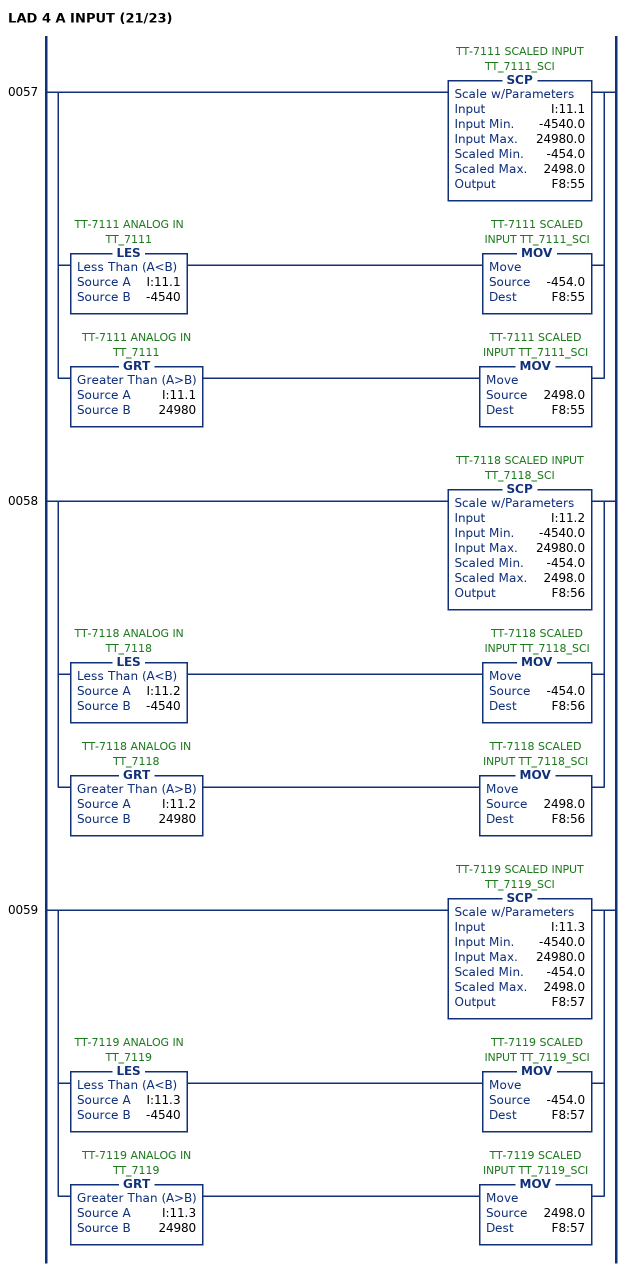
% Rung: 57 %
SOR BST SCP I:11.1 -4540.0 24980.0 -454.0 2498.0 F8:55 NXB LES I:11.1 -4540 MOV -454.0 F8:55 NXB GRT I:11.1 24980 MOV 2498.0 F8:55 BND EOR
%   I:11.1  TT_7111  "TT-7111 ANALOG IN" %
%   F8:55  TT_7111_SCI  "TT-7111 SCALED INPUT" %
% Rung: 58 %
SOR BST SCP I:11.2 -4540.0 24980.0 -454.0 2498.0 F8:56 NXB LES I:11.2 -4540 MOV -454.0 F8:56 NXB GRT I:11.2 24980 MOV 2498.0 F8:56 BND EOR
%   I:11.2  TT_7118  "TT-7118 ANALOG IN" %
%   F8:56  TT_7118_SCI  "TT-7118 SCALED INPUT" %
% Rung: 59 %
SOR BST SCP I:11.3 -4540.0 24980.0 -454.0 2498.0 F8:57 NXB LES I:11.3 -4540 MOV -454.0 F8:57 NXB GRT I:11.3 24980 MOV 2498.0 F8:57 BND EOR
%   I:11.3  TT_7119  "TT-7119 ANALOG IN" %
%   F8:57  TT_7119_SCI  "TT-7119 SCALED INPUT" %

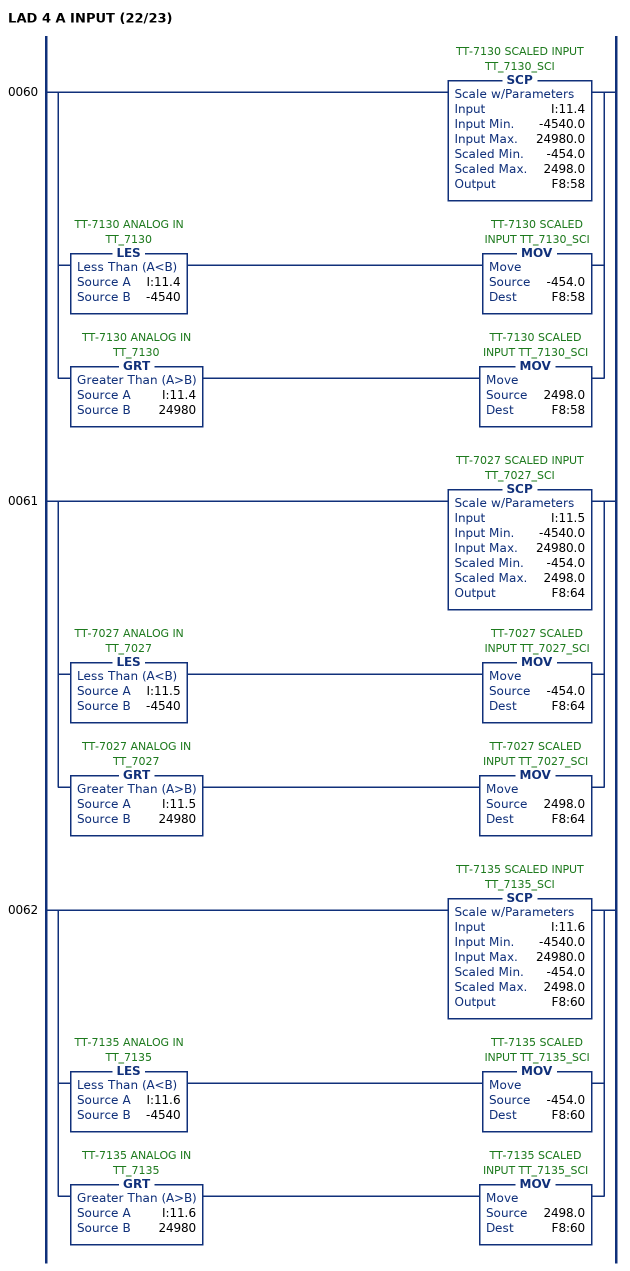
% Rung: 60 %
SOR BST SCP I:11.4 -4540.0 24980.0 -454.0 2498.0 F8:58 NXB LES I:11.4 -4540 MOV -454.0 F8:58 NXB GRT I:11.4 24980 MOV 2498.0 F8:58 BND EOR
%   I:11.4  TT_7130  "TT-7130 ANALOG IN" %
%   F8:58  TT_7130_SCI  "TT-7130 SCALED INPUT" %
% Rung: 61 %
SOR BST SCP I:11.5 -4540.0 24980.0 -454.0 2498.0 F8:64 NXB LES I:11.5 -4540 MOV -454.0 F8:64 NXB GRT I:11.5 24980 MOV 2498.0 F8:64 BND EOR
%   I:11.5  TT_7027  "TT-7027 ANALOG IN" %
%   F8:64  TT_7027_SCI  "TT-7027 SCALED INPUT" %
% Rung: 62 %
SOR BST SCP I:11.6 -4540.0 24980.0 -454.0 2498.0 F8:60 NXB LES I:11.6 -4540 MOV -454.0 F8:60 NXB GRT I:11.6 24980 MOV 2498.0 F8:60 BND EOR
%   I:11.6  TT_7135  "TT-7135 ANALOG IN" %
%   F8:60  TT_7135_SCI  "TT-7135 SCALED INPUT" %

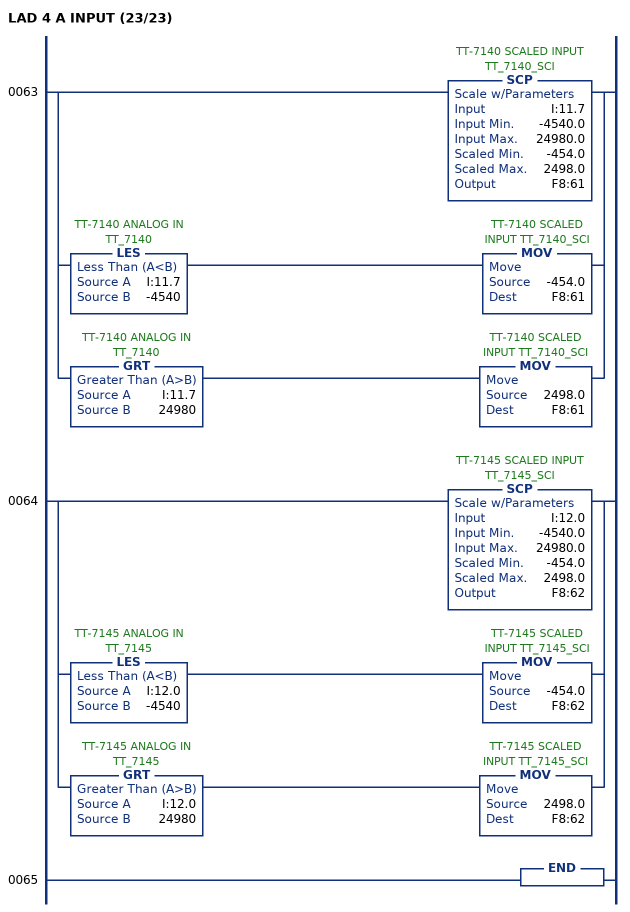
% Rung: 63 %
SOR BST SCP I:11.7 -4540.0 24980.0 -454.0 2498.0 F8:61 NXB LES I:11.7 -4540 MOV -454.0 F8:61 NXB GRT I:11.7 24980 MOV 2498.0 F8:61 BND EOR
%   I:11.7  TT_7140  "TT-7140 ANALOG IN" %
%   F8:61  TT_7140_SCI  "TT-7140 SCALED INPUT" %
% Rung: 64 %
SOR BST SCP I:12.0 -4540.0 24980.0 -454.0 2498.0 F8:62 NXB LES I:12.0 -4540 MOV -454.0 F8:62 NXB GRT I:12.0 24980 MOV 2498.0 F8:62 BND EOR
%   I:12.0  TT_7145  "TT-7145 ANALOG IN" %
%   F8:62  TT_7145_SCI  "TT-7145 SCALED INPUT" %
% Rung: 65 %
SOR END EOR

LADDER 5 "D OUTPUT"
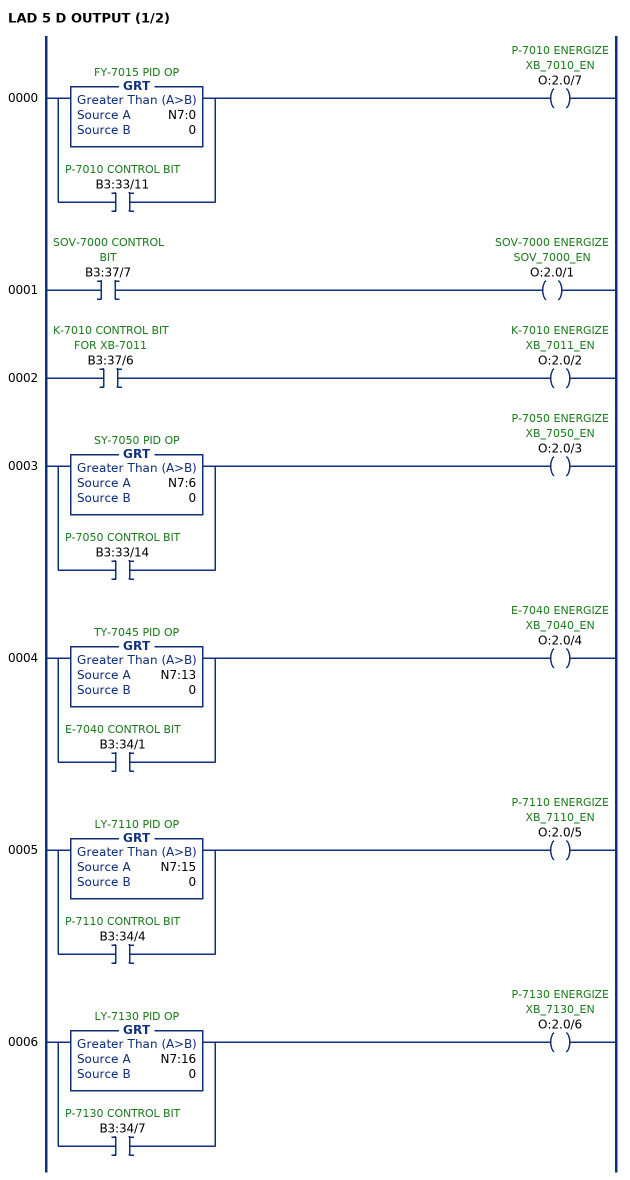
% Rung: 0 %
SOR BST GRT N7:0 0 NXB XIC B3:33/11 BND OTE O:2.0/7 EOR
%   N7:0  "FY-7015 PID OP" %
%   B3:33/11  "P-7010 CONTROL BIT" %
%   O:2.0/7  XB_7010_EN  "P-7010 ENERGIZE" %
% Rung: 1 %
SOR XIC B3:37/7 OTE O:2.0/1 EOR
%   B3:37/7  "SOV-7000 CONTROL BIT" %
%   O:2.0/1  SOV_7000_EN  "SOV-7000 ENERGIZE" %
% Rung: 2 %
SOR XIC B3:37/6 OTE O:2.0/2 EOR
%   B3:37/6  "K-7010 CONTROL BIT FOR XB-7011" %
%   O:2.0/2  XB_7011_EN  "K-7010 ENERGIZE" %
% Rung: 3 %
SOR BST GRT N7:6 0 NXB XIC B3:33/14 BND OTE O:2.0/3 EOR
%   N7:6  "SY-7050 PID OP" %
%   B3:33/14  "P-7050 CONTROL BIT" %
%   O:2.0/3  XB_7050_EN  "P-7050 ENERGIZE" %
% Rung: 4 %
SOR BST GRT N7:13 0 NXB XIC B3:34/1 BND OTE O:2.0/4 EOR
%   N7:13  "TY-7045 PID OP" %
%   B3:34/1  "E-7040 CONTROL BIT" %
%   O:2.0/4  XB_7040_EN  "E-7040 ENERGIZE" %
% Rung: 5 %
SOR BST GRT N7:15 0 NXB XIC B3:34/4 BND OTE O:2.0/5 EOR
%   N7:15  "LY-7110 PID OP" %
%   B3:34/4  "P-7110 CONTROL BIT" %
%   O:2.0/5  XB_7110_EN  "P-7110 ENERGIZE" %
% Rung: 6 %
SOR BST GRT N7:16 0 NXB XIC B3:34/7 BND OTE O:2.0/6 EOR
%   N7:16  "LY-7130 PID OP" %
%   B3:34/7  "P-7130 CONTROL BIT" %
%   O:2.0/6  XB_7130_EN  "P-7130 ENERGIZE" %

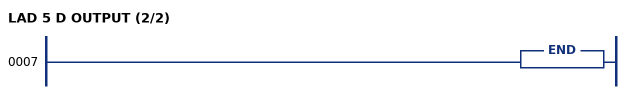
% Rung: 7 %
SOR END EOR

LADDER 6 "A OUTPUT"
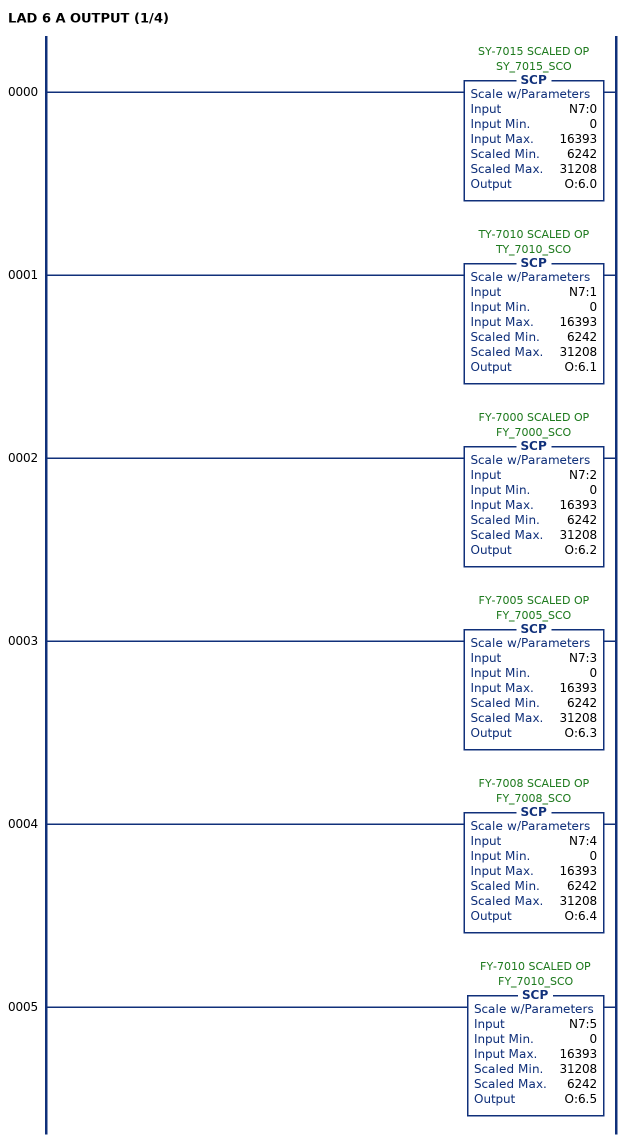
% Rung: 0 %
SOR SCP N7:0 0 16393 6242 31208 O:6.0 EOR
%   N7:0  "FY-7015 PID OP" %
%   O:6.0  SY_7015_SCO  "SY-7015 SCALED OP" %
% Rung: 1 %
SOR SCP N7:1 0 16393 6242 31208 O:6.1 EOR
%   N7:1  "TY-7010 PID OP" %
%   O:6.1  TY_7010_SCO  "TY-7010 SCALED OP" %
% Rung: 2 %
SOR SCP N7:2 0 16393 6242 31208 O:6.2 EOR
%   N7:2  "FY-7000 PID OP" %
%   O:6.2  FY_7000_SCO  "FY-7000 SCALED OP" %
% Rung: 3 %
SOR SCP N7:3 0 16393 6242 31208 O:6.3 EOR
%   N7:3  "FY-7005 PID OP" %
%   O:6.3  FY_7005_SCO  "FY-7005 SCALED OP" %
% Rung: 4 %
SOR SCP N7:4 0 16393 6242 31208 O:6.4 EOR
%   N7:4  "FY-7008 PID OP" %
%   O:6.4  FY_7008_SCO  "FY-7008 SCALED OP" %
% Rung: 5 %
SOR SCP N7:5 0 16393 31208 6242 O:6.5 EOR
%   N7:5  "FY-7010 PID OP" %
%   O:6.5  FY_7010_SCO  "FY-7010 SCALED OP" %

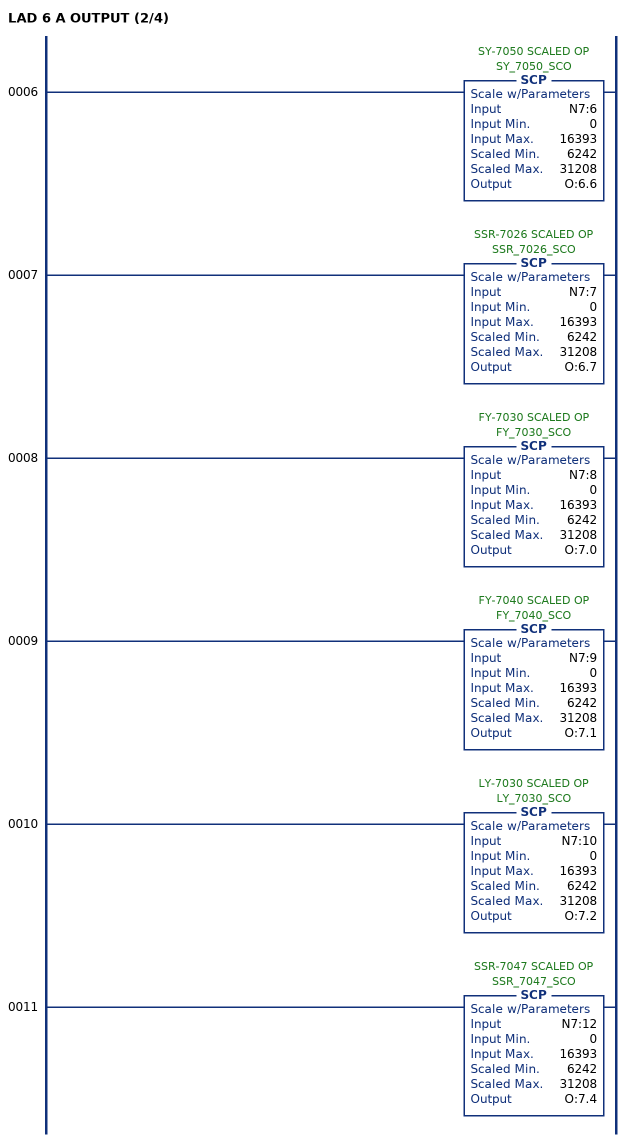
% Rung: 6 %
SOR SCP N7:6 0 16393 6242 31208 O:6.6 EOR
%   N7:6  "SY-7050 PID OP" %
%   O:6.6  SY_7050_SCO  "SY-7050 SCALED OP" %
% Rung: 7 %
SOR SCP N7:7 0 16393 6242 31208 O:6.7 EOR
%   N7:7  "SSR-7026 PID OP" %
%   O:6.7  SSR_7026_SCO  "SSR-7026 SCALED OP" %
% Rung: 8 %
SOR SCP N7:8 0 16393 6242 31208 O:7.0 EOR
%   N7:8  "FY-7030 PID OP" %
%   O:7.0  FY_7030_SCO  "FY-7030 SCALED OP" %
% Rung: 9 %
SOR SCP N7:9 0 16393 6242 31208 O:7.1 EOR
%   N7:9  "FY-7040 PID OP" %
%   O:7.1  FY_7040_SCO  "FY-7040 SCALED OP" %
% Rung: 10 %
SOR SCP N7:10 0 16393 6242 31208 O:7.2 EOR
%   N7:10  "LY-7030 PID OP" %
%   O:7.2  LY_7030_SCO  "LY-7030 SCALED OP" %
% Rung: 11 %
SOR SCP N7:12 0 16393 6242 31208 O:7.4 EOR
%   N7:12  "SSR-7047 PID OP" %
%   O:7.4  SSR_7047_SCO  "SSR-7047 SCALED OP" %

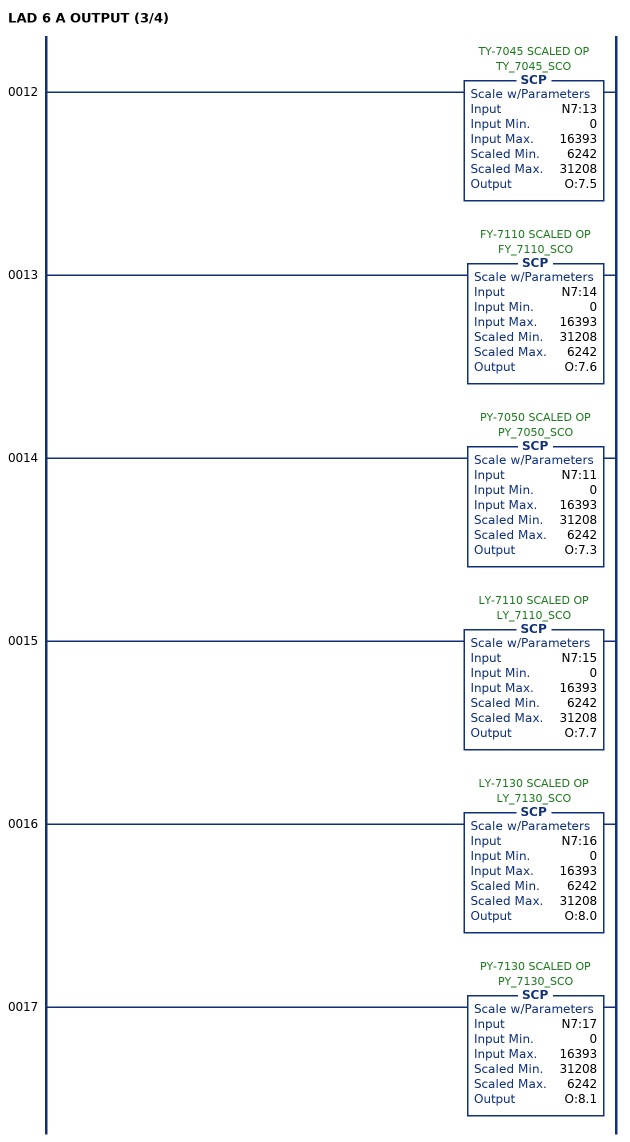
% Rung: 12 %
SOR SCP N7:13 0 16393 6242 31208 O:7.5 EOR
%   N7:13  "TY-7045 PID OP" %
%   O:7.5  TY_7045_SCO  "TY-7045 SCALED OP" %
% Rung: 13 %
SOR SCP N7:14 0 16393 31208 6242 O:7.6 EOR
%   N7:14  "FY-7110 PID OP" %
%   O:7.6  FY_7110_SCO  "FY-7110 SCALED OP" %
% Rung: 14 %
SOR SCP N7:11 0 16393 31208 6242 O:7.3 EOR
%   N7:11  "PY-7050 PID OP" %
%   O:7.3  PY_7050_SCO  "PY-7050 SCALED OP" %
% Rung: 15 %
SOR SCP N7:15 0 16393 6242 31208 O:7.7 EOR
%   N7:15  "LY-7110 PID OP" %
%   O:7.7  LY_7110_SCO  "LY-7110 SCALED OP" %
% Rung: 16 %
SOR SCP N7:16 0 16393 6242 31208 O:8.0 EOR
%   N7:16  "LY-7130 PID OP" %
%   O:8.0  LY_7130_SCO  "LY-7130 SCALED OP" %
% Rung: 17 %
SOR SCP N7:17 0 16393 31208 6242 O:8.1 EOR
%   N7:17  "PY-7130 PID OP" %
%   O:8.1  PY_7130_SCO  "PY-7130 SCALED OP" %

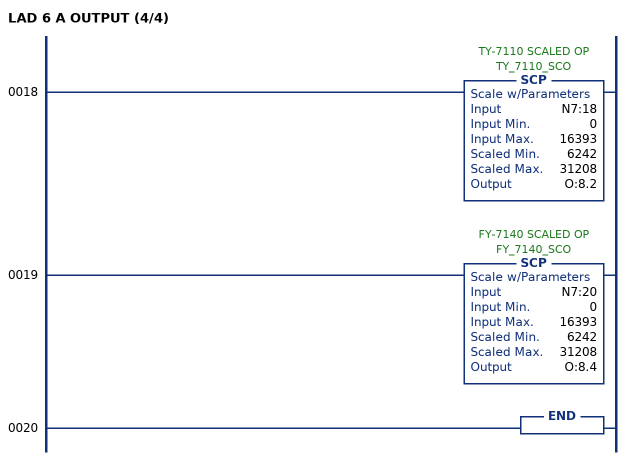
% Rung: 18 %
SOR SCP N7:18 0 16393 6242 31208 O:8.2 EOR
%   N7:18  "TY-7110 PID OP" %
%   O:8.2  TY_7110_SCO  "TY-7110 SCALED OP" %
% Rung: 19 %
SOR SCP N7:20 0 16393 6242 31208 O:8.4 EOR
%   N7:20  "FY-7140 PID OP" %
%   O:8.4  FY_7140_SCO  "FY-7140 SCALED OP" %
% Rung: 20 %
SOR END EOR

LADDER 7 "ALARMS"
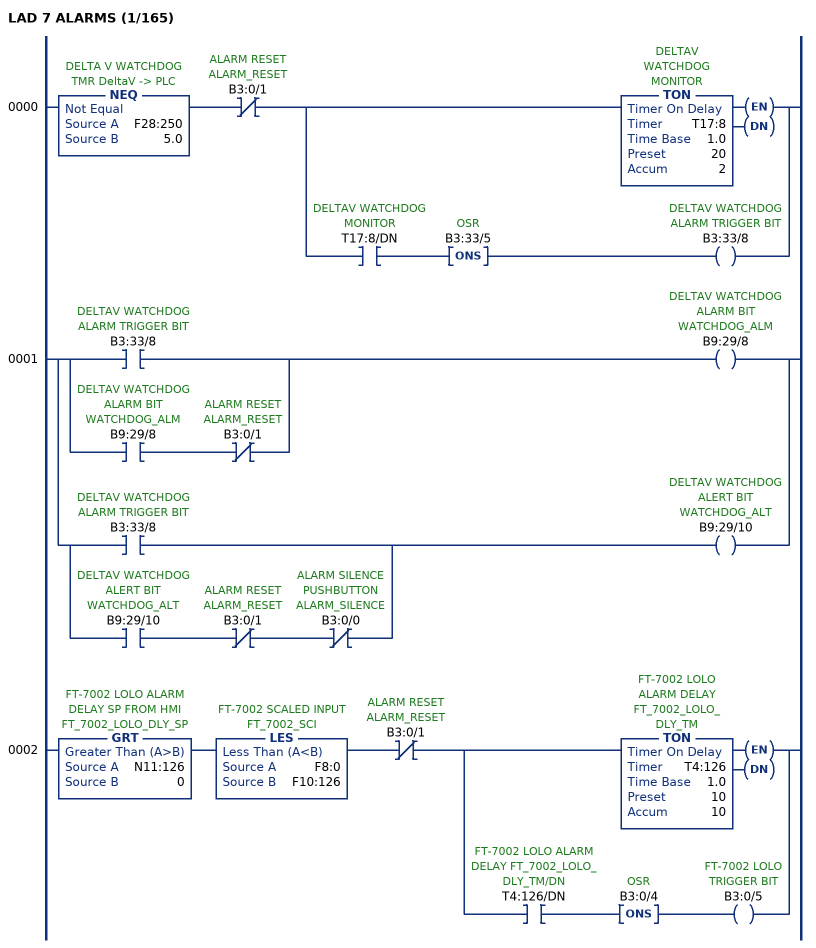
% Rung: 0 %
SOR NEQ F28:250 5.0 XIO B3:0/1 BST TON T17:8 1.0 20 2 NXB XIC T17:8/DN OSR B3:33/5 OTE B3:33/8 BND EOR
%   F28:250  "DELTA V WATCHDOG TMR DeltaV -> PLC" %
%   B3:0/1  ALARM_RESET  "ALARM RESET" %
%   T17:8  "DELTAV WATCHDOG MONITOR" %
%   B3:33/5  "OSR" %
%   B3:33/8  "DELTAV WATCHDOG ALARM TRIGGER BIT" %
% Rung: 1 %
SOR BST BST XIC B3:33/8 NXB XIC B9:29/8 XIO B3:0/1 BND OTE B9:29/8 NXB BST XIC B3:33/8 NXB XIC B9:29/10 XIO B3:0/1 XIO B3:0/0 BND OTE B9:29/10 BND EOR
%   B3:33/8  "DELTAV WATCHDOG ALARM TRIGGER BIT" %
%   B9:29/8  WATCHDOG_ALM  "DELTAV WATCHDOG ALARM BIT" %
%   B3:0/1  ALARM_RESET  "ALARM RESET" %
%   B9:29/10  WATCHDOG_ALT  "DELTAV WATCHDOG ALERT BIT" %
%   B3:0/0  ALARM_SILENCE  "ALARM SILENCE PUSHBUTTON" %
% Rung: 2 %
SOR GRT N11:126 0 LES F8:0 F10:126 XIO B3:0/1 BST TON T4:126 1.0 10 10 NXB XIC T4:126/DN OSR B3:0/4 OTE B3:0/5 BND EOR
%   N11:126  FT_7002_LOLO_DLY_SP  "FT-7002 LOLO ALARM DELAY SP FROM HMI" %
%   F8:0  FT_7002_SCI  "FT-7002 SCALED INPUT" %
%   F10:126  FT_7002_LOLO_SP  "FT-7002 LOLO ALARM SP" %
%   B3:0/1  ALARM_RESET  "ALARM RESET" %
%   T4:126  FT_7002_LOLO_DLY_TM  "FT-7002 LOLO ALARM DELAY" %
%   B3:0/4  "OSR" %
%   B3:0/5  "FT-7002 LOLO TRIGGER BIT" %

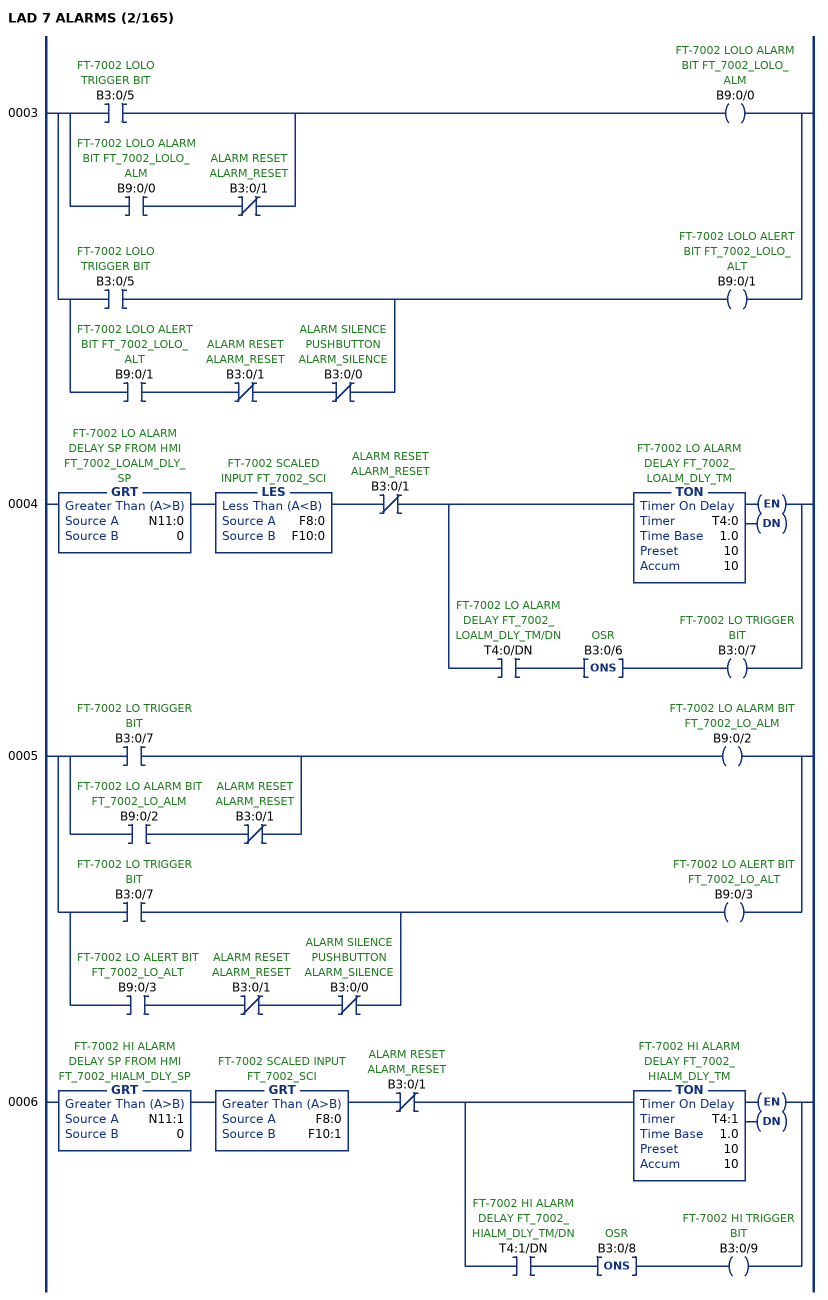
% Rung: 3 %
SOR BST BST XIC B3:0/5 NXB XIC B9:0/0 XIO B3:0/1 BND OTE B9:0/0 NXB BST XIC B3:0/5 NXB XIC B9:0/1 XIO B3:0/1 XIO B3:0/0 BND OTE B9:0/1 BND EOR
%   B3:0/5  "FT-7002 LOLO TRIGGER BIT" %
%   B9:0/0  FT_7002_LOLO_ALM  "FT-7002 LOLO ALARM BIT" %
%   B3:0/1  ALARM_RESET  "ALARM RESET" %
%   B9:0/1  FT_7002_LOLO_ALT  "FT-7002 LOLO ALERT BIT" %
%   B3:0/0  ALARM_SILENCE  "ALARM SILENCE PUSHBUTTON" %
% Rung: 4 %
SOR GRT N11:0 0 LES F8:0 F10:0 XIO B3:0/1 BST TON T4:0 1.0 10 10 NXB XIC T4:0/DN OSR B3:0/6 OTE B3:0/7 BND EOR
%   N11:0  FT_7002_LOALM_DLY_SP  "FT-7002 LO ALARM DELAY SP FROM HMI" %
%   F8:0  FT_7002_SCI  "FT-7002 SCALED INPUT" %
%   F10:0  FT_7002_LOALM_SP  "FT-7002 LO ALARM SP" %
%   B3:0/1  ALARM_RESET  "ALARM RESET" %
%   T4:0  FT_7002_LOALM_DLY_TM  "FT-7002 LO ALARM DELAY" %
%   B3:0/6  "OSR" %
%   B3:0/7  "FT-7002 LO TRIGGER BIT" %
% Rung: 5 %
SOR BST BST XIC B3:0/7 NXB XIC B9:0/2 XIO B3:0/1 BND OTE B9:0/2 NXB BST XIC B3:0/7 NXB XIC B9:0/3 XIO B3:0/1 XIO B3:0/0 BND OTE B9:0/3 BND EOR
%   B3:0/7  "FT-7002 LO TRIGGER BIT" %
%   B9:0/2  FT_7002_LO_ALM  "FT-7002 LO ALARM BIT" %
%   B3:0/1  ALARM_RESET  "ALARM RESET" %
%   B9:0/3  FT_7002_LO_ALT  "FT-7002 LO ALERT BIT" %
%   B3:0/0  ALARM_SILENCE  "ALARM SILENCE PUSHBUTTON" %
% Rung: 6 %
SOR GRT N11:1 0 GRT F8:0 F10:1 XIO B3:0/1 BST TON T4:1 1.0 10 10 NXB XIC T4:1/DN OSR B3:0/8 OTE B3:0/9 BND EOR
%   N11:1  FT_7002_HIALM_DLY_SP  "FT-7002 HI ALARM DELAY SP FROM HMI" %
%   F8:0  FT_7002_SCI  "FT-7002 SCALED INPUT" %
%   F10:1  FT_7002_HIALM_SP  "FT-7002 HI ALARM SP" %
%   B3:0/1  ALARM_RESET  "ALARM RESET" %
%   T4:1  FT_7002_HIALM_DLY_TM  "FT-7002 HI ALARM DELAY" %
%   B3:0/8  "OSR" %
%   B3:0/9  "FT-7002 HI TRIGGER BIT" %

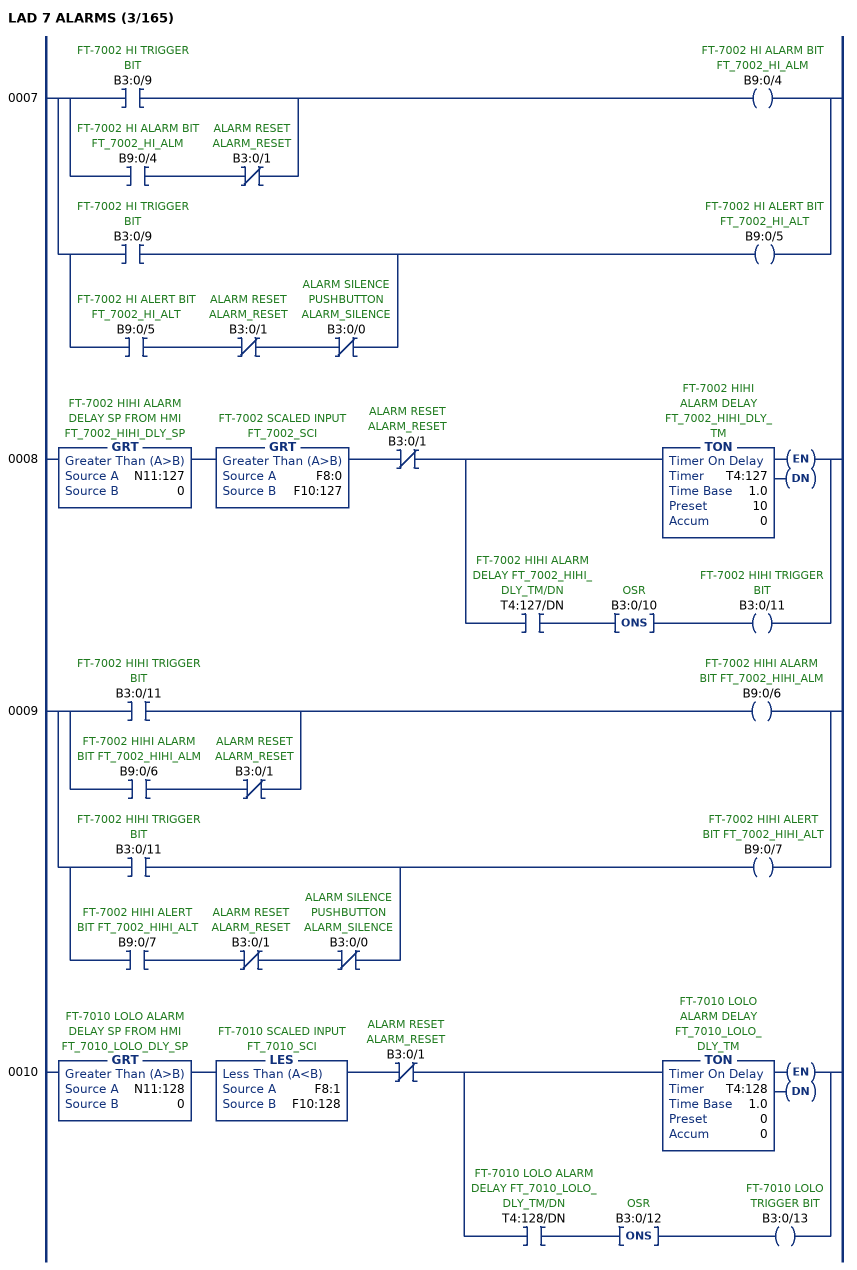
% Rung: 7 %
SOR BST BST XIC B3:0/9 NXB XIC B9:0/4 XIO B3:0/1 BND OTE B9:0/4 NXB BST XIC B3:0/9 NXB XIC B9:0/5 XIO B3:0/1 XIO B3:0/0 BND OTE B9:0/5 BND EOR
%   B3:0/9  "FT-7002 HI TRIGGER BIT" %
%   B9:0/4  FT_7002_HI_ALM  "FT-7002 HI ALARM BIT" %
%   B3:0/1  ALARM_RESET  "ALARM RESET" %
%   B9:0/5  FT_7002_HI_ALT  "FT-7002 HI ALERT BIT" %
%   B3:0/0  ALARM_SILENCE  "ALARM SILENCE PUSHBUTTON" %
% Rung: 8 %
SOR GRT N11:127 0 GRT F8:0 F10:127 XIO B3:0/1 BST TON T4:127 1.0 10 0 NXB XIC T4:127/DN OSR B3:0/10 OTE B3:0/11 BND EOR
%   N11:127  FT_7002_HIHI_DLY_SP  "FT-7002 HIHI ALARM DELAY SP FROM HMI" %
%   F8:0  FT_7002_SCI  "FT-7002 SCALED INPUT" %
%   F10:127  FT_7002_HIHI_SP  "FT-7002 HIHI ALARM SP" %
%   B3:0/1  ALARM_RESET  "ALARM RESET" %
%   T4:127  FT_7002_HIHI_DLY_TM  "FT-7002 HIHI ALARM DELAY" %
%   B3:0/10  "OSR" %
%   B3:0/11  "FT-7002 HIHI TRIGGER BIT" %
% Rung: 9 %
SOR BST BST XIC B3:0/11 NXB XIC B9:0/6 XIO B3:0/1 BND OTE B9:0/6 NXB BST XIC B3:0/11 NXB XIC B9:0/7 XIO B3:0/1 XIO B3:0/0 BND OTE B9:0/7 BND EOR
%   B3:0/11  "FT-7002 HIHI TRIGGER BIT" %
%   B9:0/6  FT_7002_HIHI_ALM  "FT-7002 HIHI ALARM BIT" %
%   B3:0/1  ALARM_RESET  "ALARM RESET" %
%   B9:0/7  FT_7002_HIHI_ALT  "FT-7002 HIHI ALERT BIT" %
%   B3:0/0  ALARM_SILENCE  "ALARM SILENCE PUSHBUTTON" %
% Rung: 10 %
SOR GRT N11:128 0 LES F8:1 F10:128 XIO B3:0/1 BST TON T4:128 1.0 0 0 NXB XIC T4:128/DN OSR B3:0/12 OTE B3:0/13 BND EOR
%   N11:128  FT_7010_LOLO_DLY_SP  "FT-7010 LOLO ALARM DELAY SP FROM HMI" %
%   F8:1  FT_7010_SCI  "FT-7010 SCALED INPUT" %
%   F10:128  FT_7010_LOLO_SP  "FT-7010 LOLO ALARM SP" %
%   B3:0/1  ALARM_RESET  "ALARM RESET" %
%   T4:128  FT_7010_LOLO_DLY_TM  "FT-7010 LOLO ALARM DELAY" %
%   B3:0/12  "OSR" %
%   B3:0/13  "FT-7010 LOLO TRIGGER BIT" %

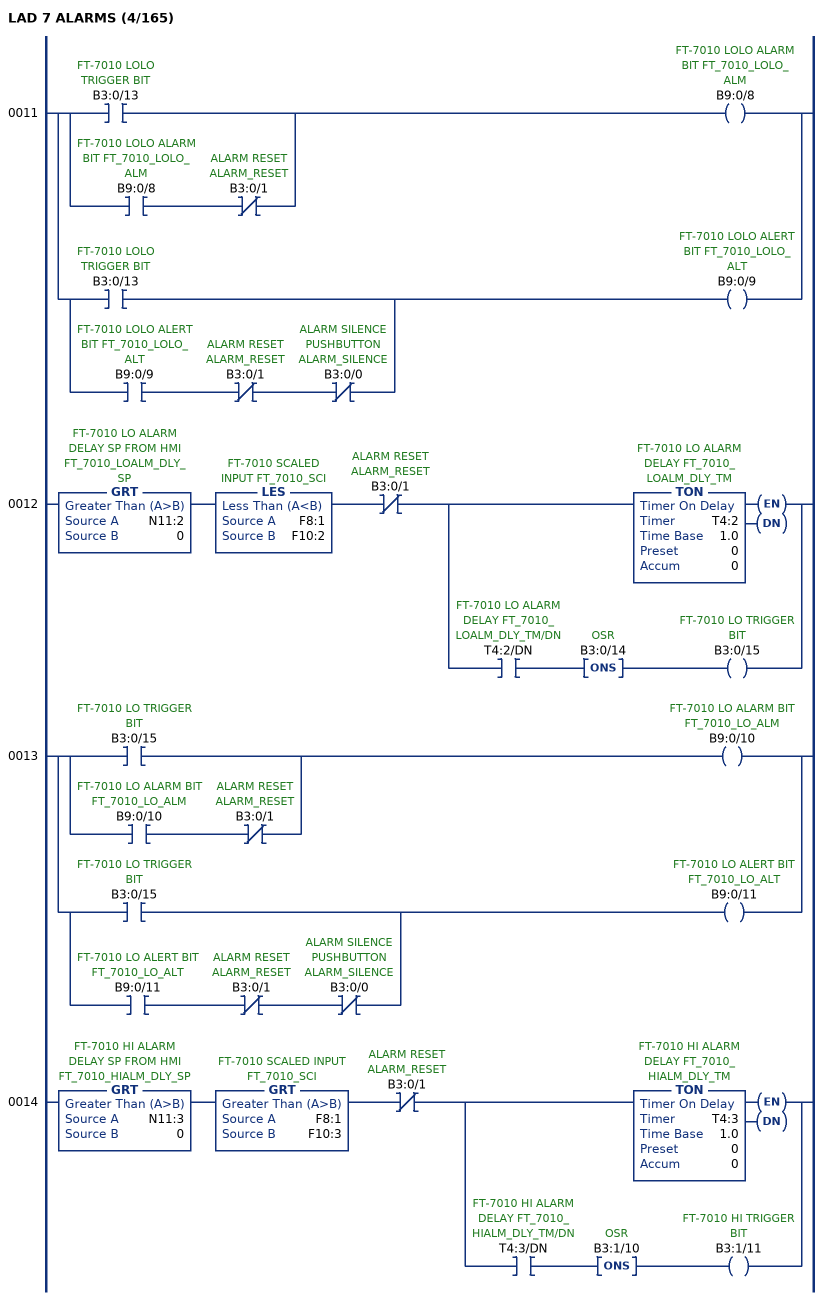
% Rung: 11 %
SOR BST BST XIC B3:0/13 NXB XIC B9:0/8 XIO B3:0/1 BND OTE B9:0/8 NXB BST XIC B3:0/13 NXB XIC B9:0/9 XIO B3:0/1 XIO B3:0/0 BND OTE B9:0/9 BND EOR
%   B3:0/13  "FT-7010 LOLO TRIGGER BIT" %
%   B9:0/8  FT_7010_LOLO_ALM  "FT-7010 LOLO ALARM BIT" %
%   B3:0/1  ALARM_RESET  "ALARM RESET" %
%   B9:0/9  FT_7010_LOLO_ALT  "FT-7010 LOLO ALERT BIT" %
%   B3:0/0  ALARM_SILENCE  "ALARM SILENCE PUSHBUTTON" %
% Rung: 12 %
SOR GRT N11:2 0 LES F8:1 F10:2 XIO B3:0/1 BST TON T4:2 1.0 0 0 NXB XIC T4:2/DN OSR B3:0/14 OTE B3:0/15 BND EOR
%   N11:2  FT_7010_LOALM_DLY_SP  "FT-7010 LO ALARM DELAY SP FROM HMI" %
%   F8:1  FT_7010_SCI  "FT-7010 SCALED INPUT" %
%   F10:2  FT_7010_LOALM_SP  "FT-7010 LO ALARM SP" %
%   B3:0/1  ALARM_RESET  "ALARM RESET" %
%   T4:2  FT_7010_LOALM_DLY_TM  "FT-7010 LO ALARM DELAY" %
%   B3:0/14  "OSR" %
%   B3:0/15  "FT-7010 LO TRIGGER BIT" %
% Rung: 13 %
SOR BST BST XIC B3:0/15 NXB XIC B9:0/10 XIO B3:0/1 BND OTE B9:0/10 NXB BST XIC B3:0/15 NXB XIC B9:0/11 XIO B3:0/1 XIO B3:0/0 BND OTE B9:0/11 BND EOR
%   B3:0/15  "FT-7010 LO TRIGGER BIT" %
%   B9:0/10  FT_7010_LO_ALM  "FT-7010 LO ALARM BIT" %
%   B3:0/1  ALARM_RESET  "ALARM RESET" %
%   B9:0/11  FT_7010_LO_ALT  "FT-7010 LO ALERT BIT" %
%   B3:0/0  ALARM_SILENCE  "ALARM SILENCE PUSHBUTTON" %
% Rung: 14 %
SOR GRT N11:3 0 GRT F8:1 F10:3 XIO B3:0/1 BST TON T4:3 1.0 0 0 NXB XIC T4:3/DN OSR B3:1/10 OTE B3:1/11 BND EOR
%   N11:3  FT_7010_HIALM_DLY_SP  "FT-7010 HI ALARM DELAY SP FROM HMI" %
%   F8:1  FT_7010_SCI  "FT-7010 SCALED INPUT" %
%   F10:3  FT_7010_HIALM_SP  "FT-7010 HI ALARM SP" %
%   B3:0/1  ALARM_RESET  "ALARM RESET" %
%   T4:3  FT_7010_HIALM_DLY_TM  "FT-7010 HI ALARM DELAY" %
%   B3:1/10  "OSR" %
%   B3:1/11  "FT-7010 HI TRIGGER BIT" %

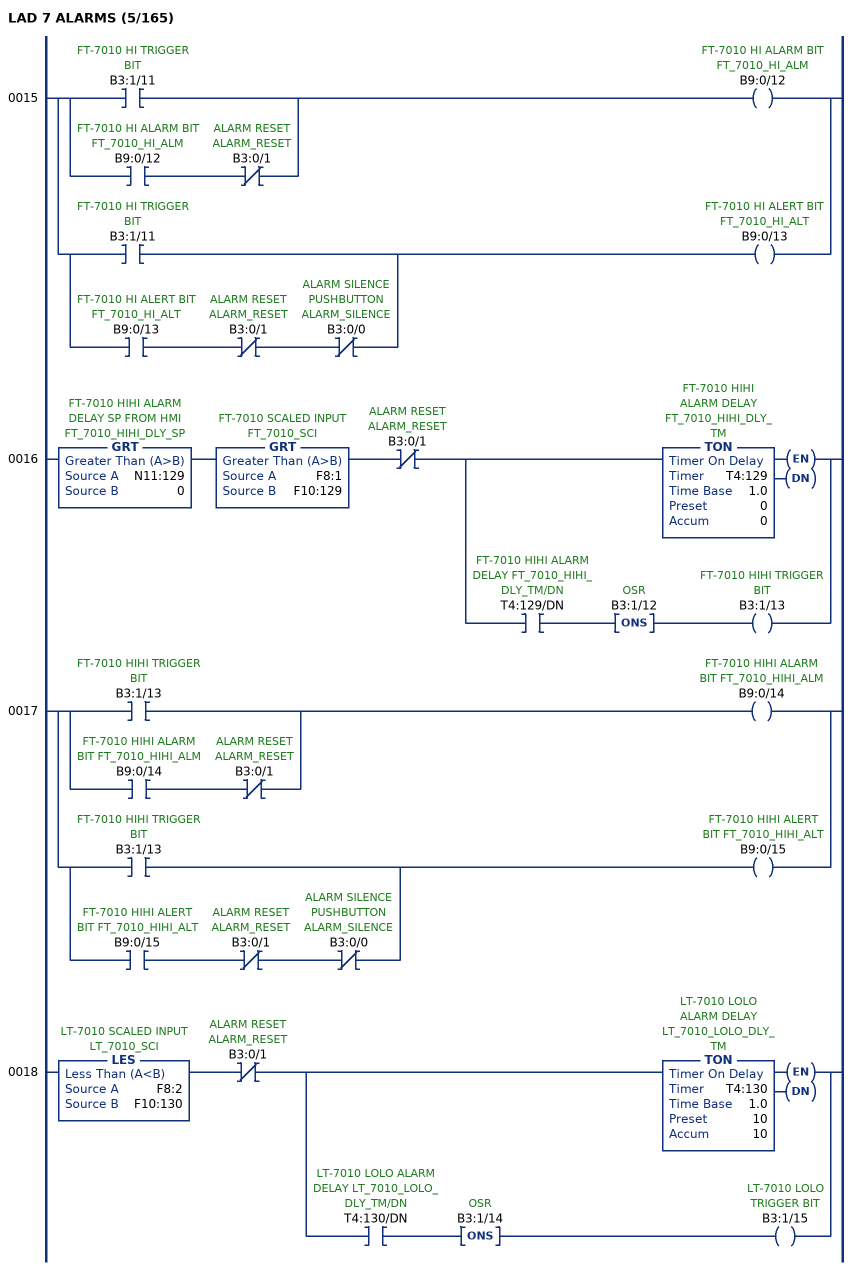
% Rung: 15 %
SOR BST BST XIC B3:1/11 NXB XIC B9:0/12 XIO B3:0/1 BND OTE B9:0/12 NXB BST XIC B3:1/11 NXB XIC B9:0/13 XIO B3:0/1 XIO B3:0/0 BND OTE B9:0/13 BND EOR
%   B3:1/11  "FT-7010 HI TRIGGER BIT" %
%   B9:0/12  FT_7010_HI_ALM  "FT-7010 HI ALARM BIT" %
%   B3:0/1  ALARM_RESET  "ALARM RESET" %
%   B9:0/13  FT_7010_HI_ALT  "FT-7010 HI ALERT BIT" %
%   B3:0/0  ALARM_SILENCE  "ALARM SILENCE PUSHBUTTON" %
% Rung: 16 %
SOR GRT N11:129 0 GRT F8:1 F10:129 XIO B3:0/1 BST TON T4:129 1.0 0 0 NXB XIC T4:129/DN OSR B3:1/12 OTE B3:1/13 BND EOR
%   N11:129  FT_7010_HIHI_DLY_SP  "FT-7010 HIHI ALARM DELAY SP FROM HMI" %
%   F8:1  FT_7010_SCI  "FT-7010 SCALED INPUT" %
%   F10:129  FT_7010_HIHI_SP  "FT-7010 HIHI ALARM SP" %
%   B3:0/1  ALARM_RESET  "ALARM RESET" %
%   T4:129  FT_7010_HIHI_DLY_TM  "FT-7010 HIHI ALARM DELAY" %
%   B3:1/12  "OSR" %
%   B3:1/13  "FT-7010 HIHI TRIGGER BIT" %
% Rung: 17 %
SOR BST BST XIC B3:1/13 NXB XIC B9:0/14 XIO B3:0/1 BND OTE B9:0/14 NXB BST XIC B3:1/13 NXB XIC B9:0/15 XIO B3:0/1 XIO B3:0/0 BND OTE B9:0/15 BND EOR
%   B3:1/13  "FT-7010 HIHI TRIGGER BIT" %
%   B9:0/14  FT_7010_HIHI_ALM  "FT-7010 HIHI ALARM BIT" %
%   B3:0/1  ALARM_RESET  "ALARM RESET" %
%   B9:0/15  FT_7010_HIHI_ALT  "FT-7010 HIHI ALERT BIT" %
%   B3:0/0  ALARM_SILENCE  "ALARM SILENCE PUSHBUTTON" %
% Rung: 18 %
SOR LES F8:2 F10:130 XIO B3:0/1 BST TON T4:130 1.0 10 10 NXB XIC T4:130/DN OSR B3:1/14 OTE B3:1/15 BND EOR
%   F8:2  LT_7010_SCI  "LT-7010 SCALED INPUT" %
%   F10:130  LT_7010_LOLO_SP  "LT-7010 LOLO ALARM SP" %
%   B3:0/1  ALARM_RESET  "ALARM RESET" %
%   T4:130  LT_7010_LOLO_DLY_TM  "LT-7010 LOLO ALARM DELAY" %
%   B3:1/14  "OSR" %
%   B3:1/15  "LT-7010 LOLO TRIGGER BIT" %

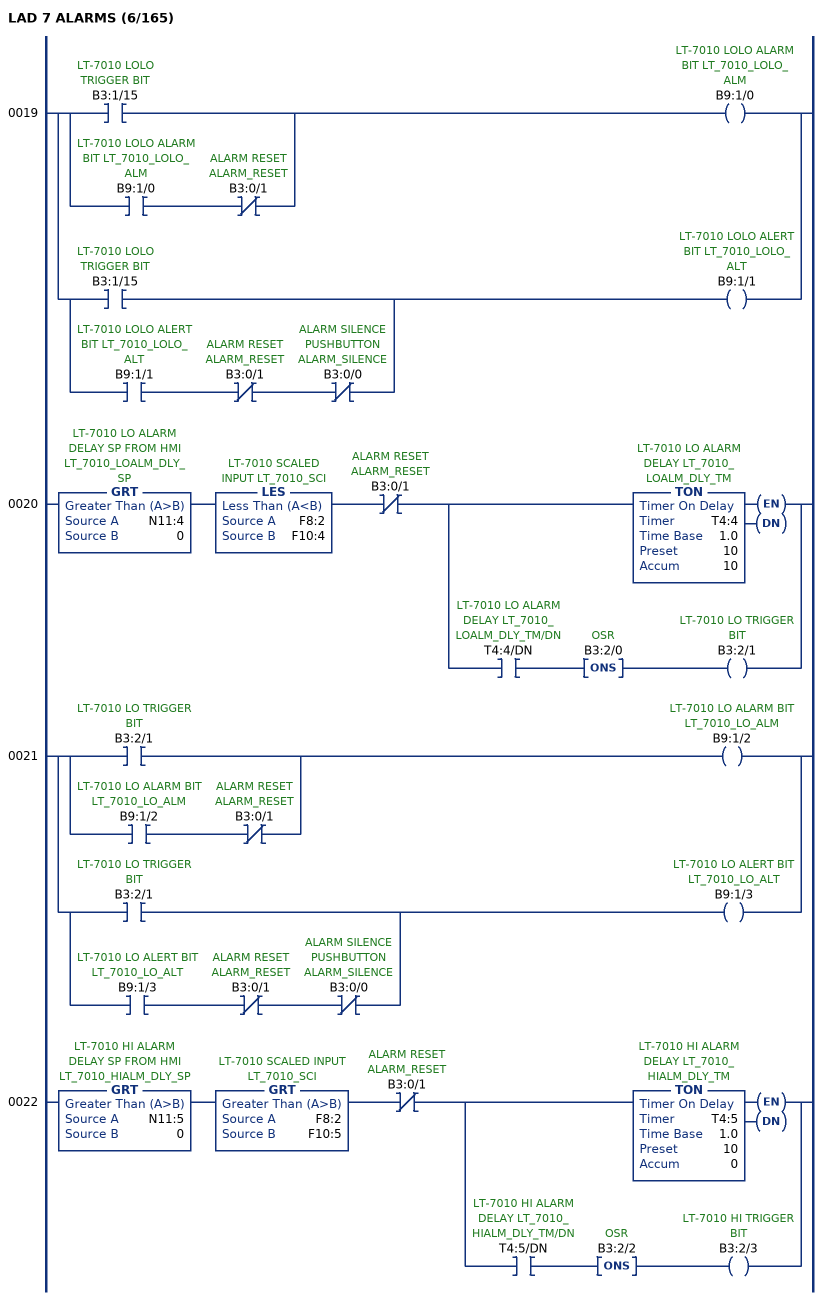
% Rung: 19 %
SOR BST BST XIC B3:1/15 NXB XIC B9:1/0 XIO B3:0/1 BND OTE B9:1/0 NXB BST XIC B3:1/15 NXB XIC B9:1/1 XIO B3:0/1 XIO B3:0/0 BND OTE B9:1/1 BND EOR
%   B3:1/15  "LT-7010 LOLO TRIGGER BIT" %
%   B9:1/0  LT_7010_LOLO_ALM  "LT-7010 LOLO ALARM BIT" %
%   B3:0/1  ALARM_RESET  "ALARM RESET" %
%   B9:1/1  LT_7010_LOLO_ALT  "LT-7010 LOLO ALERT BIT" %
%   B3:0/0  ALARM_SILENCE  "ALARM SILENCE PUSHBUTTON" %
% Rung: 20 %
SOR GRT N11:4 0 LES F8:2 F10:4 XIO B3:0/1 BST TON T4:4 1.0 10 10 NXB XIC T4:4/DN OSR B3:2/0 OTE B3:2/1 BND EOR
%   N11:4  LT_7010_LOALM_DLY_SP  "LT-7010 LO ALARM DELAY SP FROM HMI" %
%   F8:2  LT_7010_SCI  "LT-7010 SCALED INPUT" %
%   F10:4  LT_7010_LOALM_SP  "LT-7010 LO ALARM SP" %
%   B3:0/1  ALARM_RESET  "ALARM RESET" %
%   T4:4  LT_7010_LOALM_DLY_TM  "LT-7010 LO ALARM DELAY" %
%   B3:2/0  "OSR" %
%   B3:2/1  "LT-7010 LO TRIGGER BIT" %
% Rung: 21 %
SOR BST BST XIC B3:2/1 NXB XIC B9:1/2 XIO B3:0/1 BND OTE B9:1/2 NXB BST XIC B3:2/1 NXB XIC B9:1/3 XIO B3:0/1 XIO B3:0/0 BND OTE B9:1/3 BND EOR
%   B3:2/1  "LT-7010 LO TRIGGER BIT" %
%   B9:1/2  LT_7010_LO_ALM  "LT-7010 LO ALARM BIT" %
%   B3:0/1  ALARM_RESET  "ALARM RESET" %
%   B9:1/3  LT_7010_LO_ALT  "LT-7010 LO ALERT BIT" %
%   B3:0/0  ALARM_SILENCE  "ALARM SILENCE PUSHBUTTON" %
% Rung: 22 %
SOR GRT N11:5 0 GRT F8:2 F10:5 XIO B3:0/1 BST TON T4:5 1.0 10 0 NXB XIC T4:5/DN OSR B3:2/2 OTE B3:2/3 BND EOR
%   N11:5  LT_7010_HIALM_DLY_SP  "LT-7010 HI ALARM DELAY SP FROM HMI" %
%   F8:2  LT_7010_SCI  "LT-7010 SCALED INPUT" %
%   F10:5  LT_7010_HIALM_SP  "LT-7010 HI ALARM SP" %
%   B3:0/1  ALARM_RESET  "ALARM RESET" %
%   T4:5  LT_7010_HIALM_DLY_TM  "LT-7010 HI ALARM DELAY" %
%   B3:2/2  "OSR" %
%   B3:2/3  "LT-7010 HI TRIGGER BIT" %

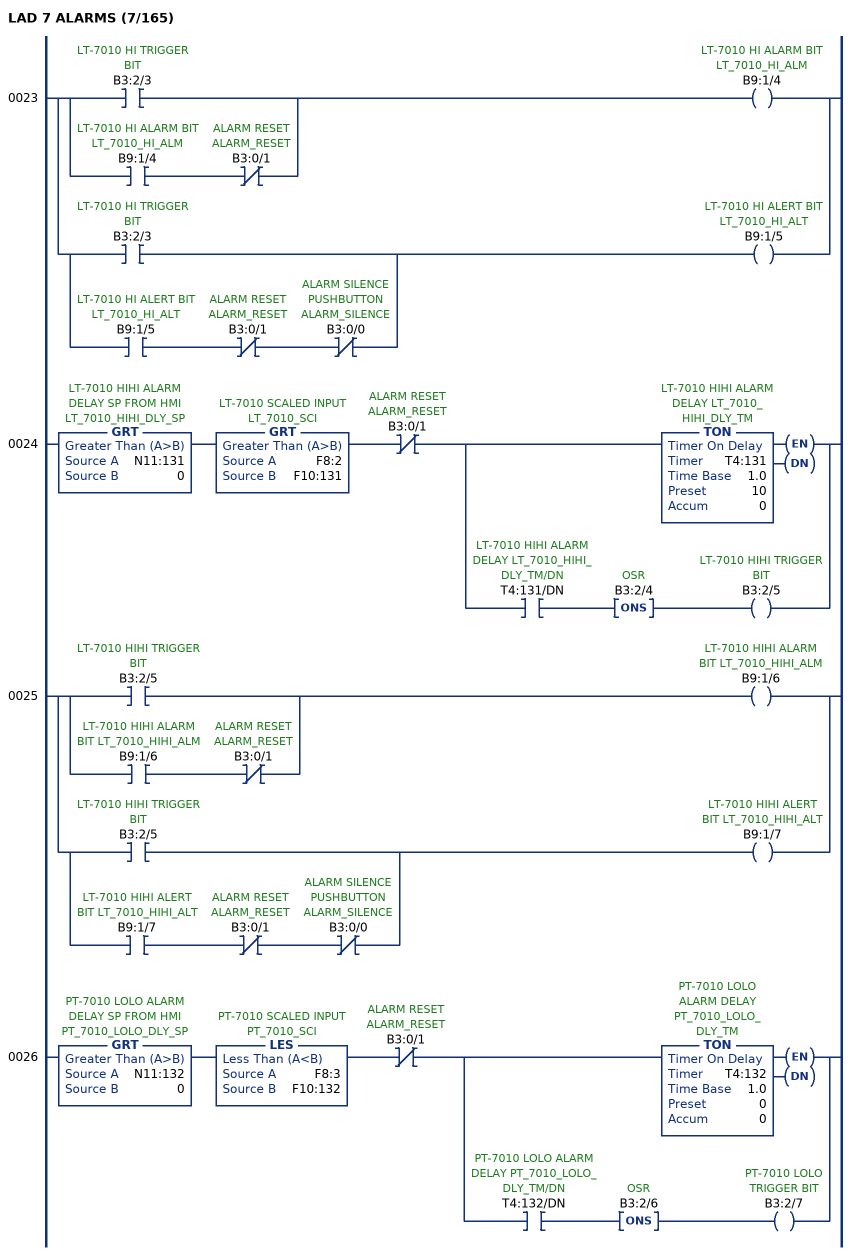
% Rung: 23 %
SOR BST BST XIC B3:2/3 NXB XIC B9:1/4 XIO B3:0/1 BND OTE B9:1/4 NXB BST XIC B3:2/3 NXB XIC B9:1/5 XIO B3:0/1 XIO B3:0/0 BND OTE B9:1/5 BND EOR
%   B3:2/3  "LT-7010 HI TRIGGER BIT" %
%   B9:1/4  LT_7010_HI_ALM  "LT-7010 HI ALARM BIT" %
%   B3:0/1  ALARM_RESET  "ALARM RESET" %
%   B9:1/5  LT_7010_HI_ALT  "LT-7010 HI ALERT BIT" %
%   B3:0/0  ALARM_SILENCE  "ALARM SILENCE PUSHBUTTON" %
% Rung: 24 %
SOR GRT N11:131 0 GRT F8:2 F10:131 XIO B3:0/1 BST TON T4:131 1.0 10 0 NXB XIC T4:131/DN OSR B3:2/4 OTE B3:2/5 BND EOR
%   N11:131  LT_7010_HIHI_DLY_SP  "LT-7010 HIHI ALARM DELAY SP FROM HMI" %
%   F8:2  LT_7010_SCI  "LT-7010 SCALED INPUT" %
%   F10:131  LT_7010_HIHI_SP  "LT-7010 HIHI ALARM SP" %
%   B3:0/1  ALARM_RESET  "ALARM RESET" %
%   T4:131  LT_7010_HIHI_DLY_TM  "LT-7010 HIHI ALARM DELAY" %
%   B3:2/4  "OSR" %
%   B3:2/5  "LT-7010 HIHI TRIGGER BIT" %
% Rung: 25 %
SOR BST BST XIC B3:2/5 NXB XIC B9:1/6 XIO B3:0/1 BND OTE B9:1/6 NXB BST XIC B3:2/5 NXB XIC B9:1/7 XIO B3:0/1 XIO B3:0/0 BND OTE B9:1/7 BND EOR
%   B3:2/5  "LT-7010 HIHI TRIGGER BIT" %
%   B9:1/6  LT_7010_HIHI_ALM  "LT-7010 HIHI ALARM BIT" %
%   B3:0/1  ALARM_RESET  "ALARM RESET" %
%   B9:1/7  LT_7010_HIHI_ALT  "LT-7010 HIHI ALERT BIT" %
%   B3:0/0  ALARM_SILENCE  "ALARM SILENCE PUSHBUTTON" %
% Rung: 26 %
SOR GRT N11:132 0 LES F8:3 F10:132 XIO B3:0/1 BST TON T4:132 1.0 0 0 NXB XIC T4:132/DN OSR B3:2/6 OTE B3:2/7 BND EOR
%   N11:132  PT_7010_LOLO_DLY_SP  "PT-7010 LOLO ALARM DELAY SP FROM HMI" %
%   F8:3  PT_7010_SCI  "PT-7010 SCALED INPUT" %
%   F10:132  PT_7010_LOLO_SP  "PT-7010 LOLO ALARM SP" %
%   B3:0/1  ALARM_RESET  "ALARM RESET" %
%   T4:132  PT_7010_LOLO_DLY_TM  "PT-7010 LOLO ALARM DELAY" %
%   B3:2/6  "OSR" %
%   B3:2/7  "PT-7010 LOLO TRIGGER BIT" %

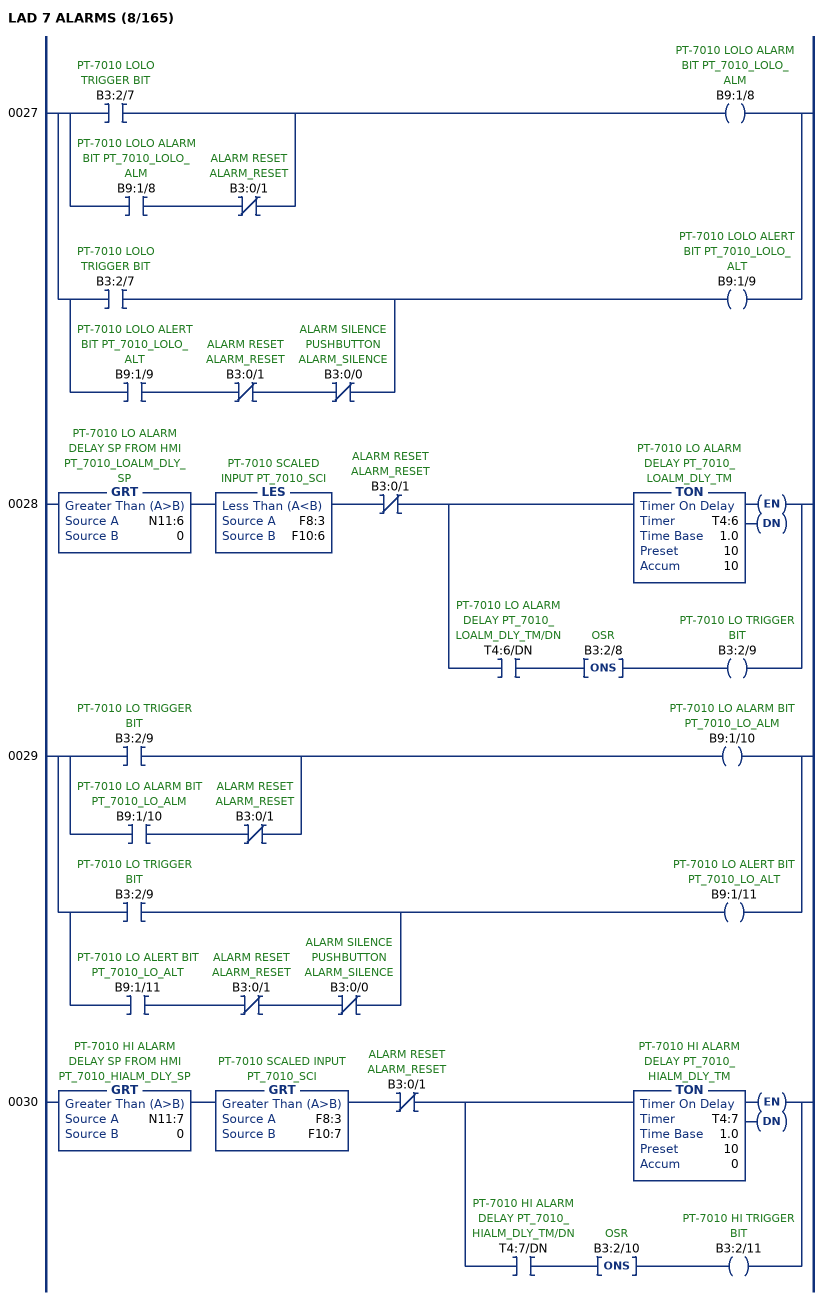
% Rung: 27 %
SOR BST BST XIC B3:2/7 NXB XIC B9:1/8 XIO B3:0/1 BND OTE B9:1/8 NXB BST XIC B3:2/7 NXB XIC B9:1/9 XIO B3:0/1 XIO B3:0/0 BND OTE B9:1/9 BND EOR
%   B3:2/7  "PT-7010 LOLO TRIGGER BIT" %
%   B9:1/8  PT_7010_LOLO_ALM  "PT-7010 LOLO ALARM BIT" %
%   B3:0/1  ALARM_RESET  "ALARM RESET" %
%   B9:1/9  PT_7010_LOLO_ALT  "PT-7010 LOLO ALERT BIT" %
%   B3:0/0  ALARM_SILENCE  "ALARM SILENCE PUSHBUTTON" %
% Rung: 28 %
SOR GRT N11:6 0 LES F8:3 F10:6 XIO B3:0/1 BST TON T4:6 1.0 10 10 NXB XIC T4:6/DN OSR B3:2/8 OTE B3:2/9 BND EOR
%   N11:6  PT_7010_LOALM_DLY_SP  "PT-7010 LO ALARM DELAY SP FROM HMI" %
%   F8:3  PT_7010_SCI  "PT-7010 SCALED INPUT" %
%   F10:6  PT_7010_LOALM_SP  "PT-7010 LO ALARM SP" %
%   B3:0/1  ALARM_RESET  "ALARM RESET" %
%   T4:6  PT_7010_LOALM_DLY_TM  "PT-7010 LO ALARM DELAY" %
%   B3:2/8  "OSR" %
%   B3:2/9  "PT-7010 LO TRIGGER BIT" %
% Rung: 29 %
SOR BST BST XIC B3:2/9 NXB XIC B9:1/10 XIO B3:0/1 BND OTE B9:1/10 NXB BST XIC B3:2/9 NXB XIC B9:1/11 XIO B3:0/1 XIO B3:0/0 BND OTE B9:1/11 BND EOR
%   B3:2/9  "PT-7010 LO TRIGGER BIT" %
%   B9:1/10  PT_7010_LO_ALM  "PT-7010 LO ALARM BIT" %
%   B3:0/1  ALARM_RESET  "ALARM RESET" %
%   B9:1/11  PT_7010_LO_ALT  "PT-7010 LO ALERT BIT" %
%   B3:0/0  ALARM_SILENCE  "ALARM SILENCE PUSHBUTTON" %
% Rung: 30 %
SOR GRT N11:7 0 GRT F8:3 F10:7 XIO B3:0/1 BST TON T4:7 1.0 10 0 NXB XIC T4:7/DN OSR B3:2/10 OTE B3:2/11 BND EOR
%   N11:7  PT_7010_HIALM_DLY_SP  "PT-7010 HI ALARM DELAY SP FROM HMI" %
%   F8:3  PT_7010_SCI  "PT-7010 SCALED INPUT" %
%   F10:7  PT_7010_HIALM_SP  "PT-7010 HI ALARM SP" %
%   B3:0/1  ALARM_RESET  "ALARM RESET" %
%   T4:7  PT_7010_HIALM_DLY_TM  "PT-7010 HI ALARM DELAY" %
%   B3:2/10  "OSR" %
%   B3:2/11  "PT-7010 HI TRIGGER BIT" %

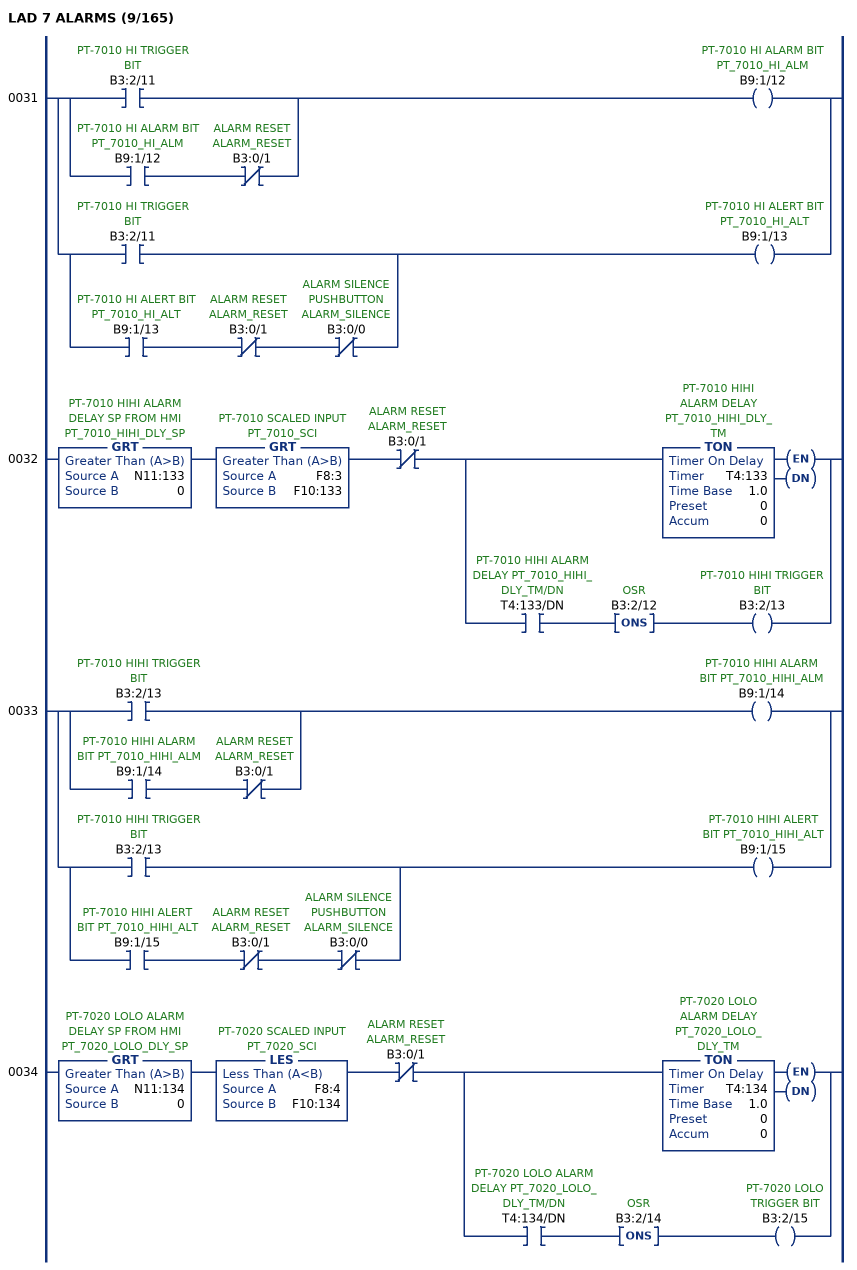
% Rung: 31 %
SOR BST BST XIC B3:2/11 NXB XIC B9:1/12 XIO B3:0/1 BND OTE B9:1/12 NXB BST XIC B3:2/11 NXB XIC B9:1/13 XIO B3:0/1 XIO B3:0/0 BND OTE B9:1/13 BND EOR
%   B3:2/11  "PT-7010 HI TRIGGER BIT" %
%   B9:1/12  PT_7010_HI_ALM  "PT-7010 HI ALARM BIT" %
%   B3:0/1  ALARM_RESET  "ALARM RESET" %
%   B9:1/13  PT_7010_HI_ALT  "PT-7010 HI ALERT BIT" %
%   B3:0/0  ALARM_SILENCE  "ALARM SILENCE PUSHBUTTON" %
% Rung: 32 %
SOR GRT N11:133 0 GRT F8:3 F10:133 XIO B3:0/1 BST TON T4:133 1.0 0 0 NXB XIC T4:133/DN OSR B3:2/12 OTE B3:2/13 BND EOR
%   N11:133  PT_7010_HIHI_DLY_SP  "PT-7010 HIHI ALARM DELAY SP FROM HMI" %
%   F8:3  PT_7010_SCI  "PT-7010 SCALED INPUT" %
%   F10:133  PT_7010_HIHI_SP  "PT-7010 HIHI ALARM SP" %
%   B3:0/1  ALARM_RESET  "ALARM RESET" %
%   T4:133  PT_7010_HIHI_DLY_TM  "PT-7010 HIHI ALARM DELAY" %
%   B3:2/12  "OSR" %
%   B3:2/13  "PT-7010 HIHI TRIGGER BIT" %
% Rung: 33 %
SOR BST BST XIC B3:2/13 NXB XIC B9:1/14 XIO B3:0/1 BND OTE B9:1/14 NXB BST XIC B3:2/13 NXB XIC B9:1/15 XIO B3:0/1 XIO B3:0/0 BND OTE B9:1/15 BND EOR
%   B3:2/13  "PT-7010 HIHI TRIGGER BIT" %
%   B9:1/14  PT_7010_HIHI_ALM  "PT-7010 HIHI ALARM BIT" %
%   B3:0/1  ALARM_RESET  "ALARM RESET" %
%   B9:1/15  PT_7010_HIHI_ALT  "PT-7010 HIHI ALERT BIT" %
%   B3:0/0  ALARM_SILENCE  "ALARM SILENCE PUSHBUTTON" %
% Rung: 34 %
SOR GRT N11:134 0 LES F8:4 F10:134 XIO B3:0/1 BST TON T4:134 1.0 0 0 NXB XIC T4:134/DN OSR B3:2/14 OTE B3:2/15 BND EOR
%   N11:134  PT_7020_LOLO_DLY_SP  "PT-7020 LOLO ALARM DELAY SP FROM HMI" %
%   F8:4  PT_7020_SCI  "PT-7020 SCALED INPUT" %
%   F10:134  PT_7020_LOLO_SP  "PT-7020 LOLO ALARM SP" %
%   B3:0/1  ALARM_RESET  "ALARM RESET" %
%   T4:134  PT_7020_LOLO_DLY_TM  "PT-7020 LOLO ALARM DELAY" %
%   B3:2/14  "OSR" %
%   B3:2/15  "PT-7020 LOLO TRIGGER BIT" %

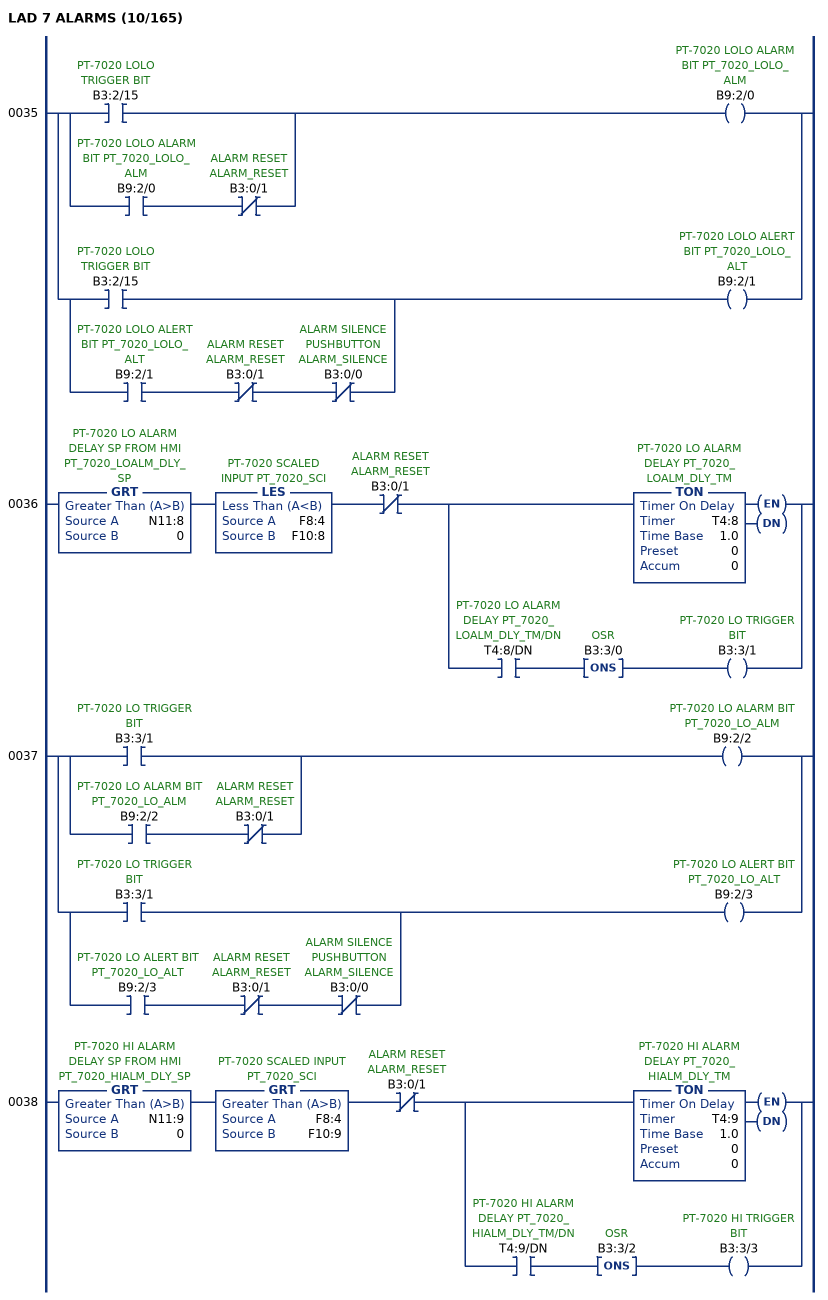
% Rung: 35 %
SOR BST BST XIC B3:2/15 NXB XIC B9:2/0 XIO B3:0/1 BND OTE B9:2/0 NXB BST XIC B3:2/15 NXB XIC B9:2/1 XIO B3:0/1 XIO B3:0/0 BND OTE B9:2/1 BND EOR
%   B3:2/15  "PT-7020 LOLO TRIGGER BIT" %
%   B9:2/0  PT_7020_LOLO_ALM  "PT-7020 LOLO ALARM BIT" %
%   B3:0/1  ALARM_RESET  "ALARM RESET" %
%   B9:2/1  PT_7020_LOLO_ALT  "PT-7020 LOLO ALERT BIT" %
%   B3:0/0  ALARM_SILENCE  "ALARM SILENCE PUSHBUTTON" %
% Rung: 36 %
SOR GRT N11:8 0 LES F8:4 F10:8 XIO B3:0/1 BST TON T4:8 1.0 0 0 NXB XIC T4:8/DN OSR B3:3/0 OTE B3:3/1 BND EOR
%   N11:8  PT_7020_LOALM_DLY_SP  "PT-7020 LO ALARM DELAY SP FROM HMI" %
%   F8:4  PT_7020_SCI  "PT-7020 SCALED INPUT" %
%   F10:8  PT_7020_LOALM_SP  "PT-7020 LO ALARM SP" %
%   B3:0/1  ALARM_RESET  "ALARM RESET" %
%   T4:8  PT_7020_LOALM_DLY_TM  "PT-7020 LO ALARM DELAY" %
%   B3:3/0  "OSR" %
%   B3:3/1  "PT-7020 LO TRIGGER BIT" %
% Rung: 37 %
SOR BST BST XIC B3:3/1 NXB XIC B9:2/2 XIO B3:0/1 BND OTE B9:2/2 NXB BST XIC B3:3/1 NXB XIC B9:2/3 XIO B3:0/1 XIO B3:0/0 BND OTE B9:2/3 BND EOR
%   B3:3/1  "PT-7020 LO TRIGGER BIT" %
%   B9:2/2  PT_7020_LO_ALM  "PT-7020 LO ALARM BIT" %
%   B3:0/1  ALARM_RESET  "ALARM RESET" %
%   B9:2/3  PT_7020_LO_ALT  "PT-7020 LO ALERT BIT" %
%   B3:0/0  ALARM_SILENCE  "ALARM SILENCE PUSHBUTTON" %
% Rung: 38 %
SOR GRT N11:9 0 GRT F8:4 F10:9 XIO B3:0/1 BST TON T4:9 1.0 0 0 NXB XIC T4:9/DN OSR B3:3/2 OTE B3:3/3 BND EOR
%   N11:9  PT_7020_HIALM_DLY_SP  "PT-7020 HI ALARM DELAY SP FROM HMI" %
%   F8:4  PT_7020_SCI  "PT-7020 SCALED INPUT" %
%   F10:9  PT_7020_HIALM_SP  "PT-7020 HI ALARM SP" %
%   B3:0/1  ALARM_RESET  "ALARM RESET" %
%   T4:9  PT_7020_HIALM_DLY_TM  "PT-7020 HI ALARM DELAY" %
%   B3:3/2  "OSR" %
%   B3:3/3  "PT-7020 HI TRIGGER BIT" %

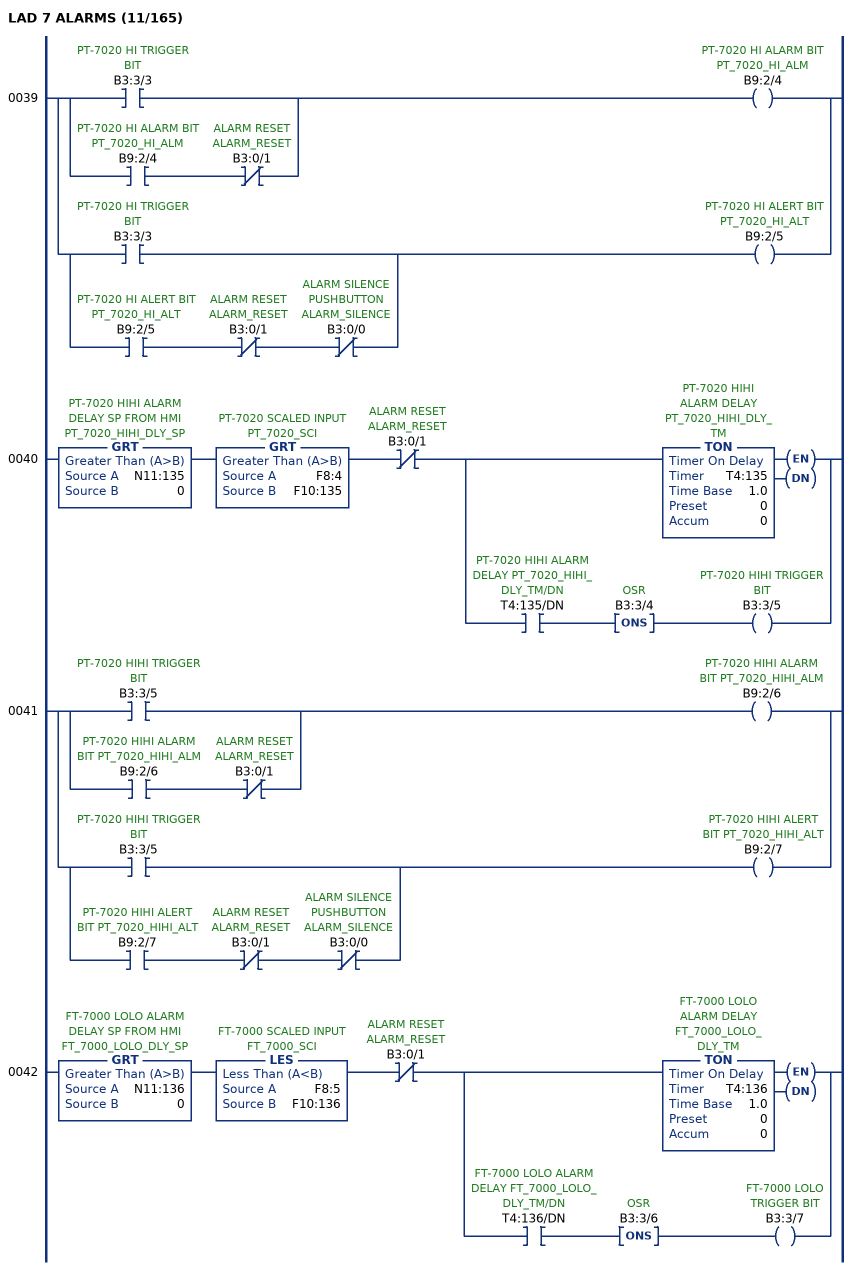
% Rung: 39 %
SOR BST BST XIC B3:3/3 NXB XIC B9:2/4 XIO B3:0/1 BND OTE B9:2/4 NXB BST XIC B3:3/3 NXB XIC B9:2/5 XIO B3:0/1 XIO B3:0/0 BND OTE B9:2/5 BND EOR
%   B3:3/3  "PT-7020 HI TRIGGER BIT" %
%   B9:2/4  PT_7020_HI_ALM  "PT-7020 HI ALARM BIT" %
%   B3:0/1  ALARM_RESET  "ALARM RESET" %
%   B9:2/5  PT_7020_HI_ALT  "PT-7020 HI ALERT BIT" %
%   B3:0/0  ALARM_SILENCE  "ALARM SILENCE PUSHBUTTON" %
% Rung: 40 %
SOR GRT N11:135 0 GRT F8:4 F10:135 XIO B3:0/1 BST TON T4:135 1.0 0 0 NXB XIC T4:135/DN OSR B3:3/4 OTE B3:3/5 BND EOR
%   N11:135  PT_7020_HIHI_DLY_SP  "PT-7020 HIHI ALARM DELAY SP FROM HMI" %
%   F8:4  PT_7020_SCI  "PT-7020 SCALED INPUT" %
%   F10:135  PT_7020_HIHI_SP  "PT-7020 HIHI ALARM SP" %
%   B3:0/1  ALARM_RESET  "ALARM RESET" %
%   T4:135  PT_7020_HIHI_DLY_TM  "PT-7020 HIHI ALARM DELAY" %
%   B3:3/4  "OSR" %
%   B3:3/5  "PT-7020 HIHI TRIGGER BIT" %
% Rung: 41 %
SOR BST BST XIC B3:3/5 NXB XIC B9:2/6 XIO B3:0/1 BND OTE B9:2/6 NXB BST XIC B3:3/5 NXB XIC B9:2/7 XIO B3:0/1 XIO B3:0/0 BND OTE B9:2/7 BND EOR
%   B3:3/5  "PT-7020 HIHI TRIGGER BIT" %
%   B9:2/6  PT_7020_HIHI_ALM  "PT-7020 HIHI ALARM BIT" %
%   B3:0/1  ALARM_RESET  "ALARM RESET" %
%   B9:2/7  PT_7020_HIHI_ALT  "PT-7020 HIHI ALERT BIT" %
%   B3:0/0  ALARM_SILENCE  "ALARM SILENCE PUSHBUTTON" %
% Rung: 42 %
SOR GRT N11:136 0 LES F8:5 F10:136 XIO B3:0/1 BST TON T4:136 1.0 0 0 NXB XIC T4:136/DN OSR B3:3/6 OTE B3:3/7 BND EOR
%   N11:136  FT_7000_LOLO_DLY_SP  "FT-7000 LOLO ALARM DELAY SP FROM HMI" %
%   F8:5  FT_7000_SCI  "FT-7000 SCALED INPUT" %
%   F10:136  FT_7000_LOLO_SP  "FT-7000 LOLO ALARM SP" %
%   B3:0/1  ALARM_RESET  "ALARM RESET" %
%   T4:136  FT_7000_LOLO_DLY_TM  "FT-7000 LOLO ALARM DELAY" %
%   B3:3/6  "OSR" %
%   B3:3/7  "FT-7000 LOLO TRIGGER BIT" %

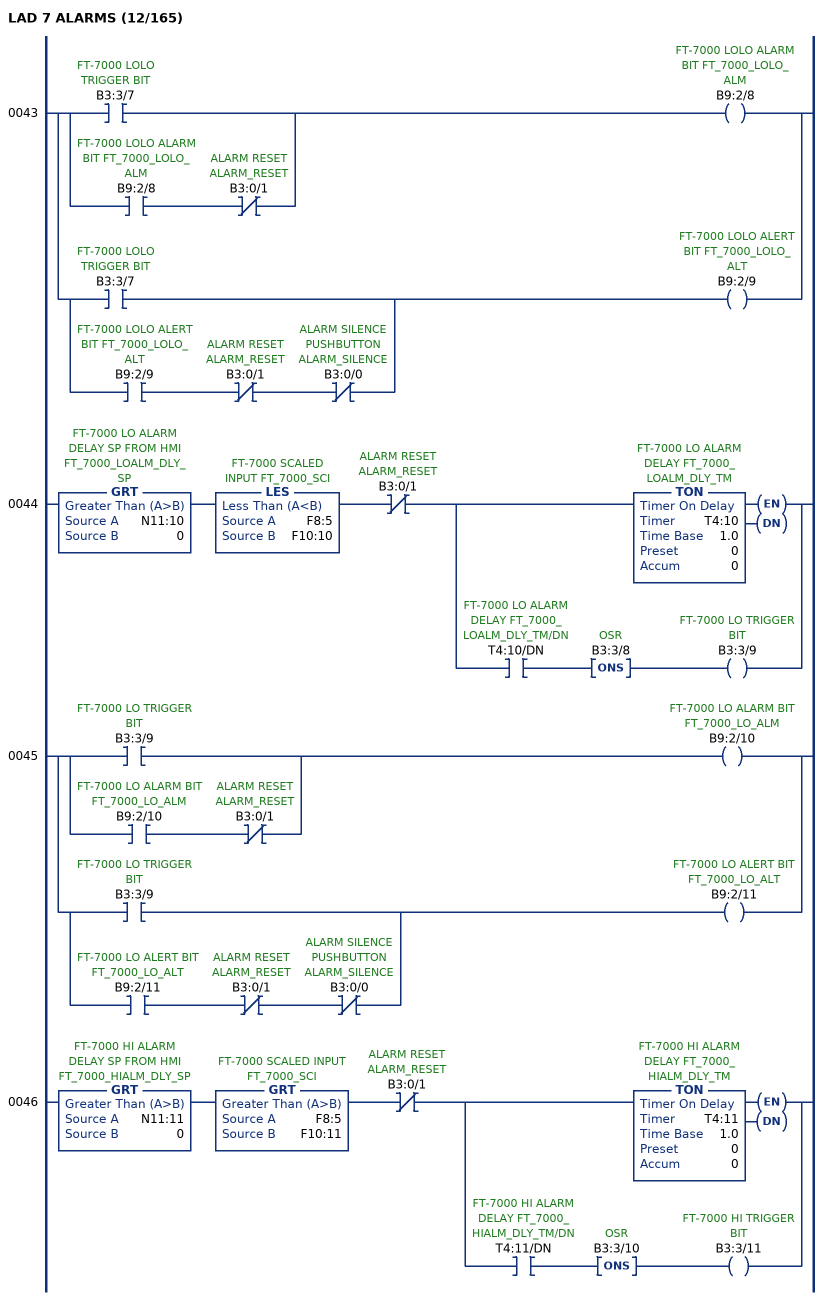
% Rung: 43 %
SOR BST BST XIC B3:3/7 NXB XIC B9:2/8 XIO B3:0/1 BND OTE B9:2/8 NXB BST XIC B3:3/7 NXB XIC B9:2/9 XIO B3:0/1 XIO B3:0/0 BND OTE B9:2/9 BND EOR
%   B3:3/7  "FT-7000 LOLO TRIGGER BIT" %
%   B9:2/8  FT_7000_LOLO_ALM  "FT-7000 LOLO ALARM BIT" %
%   B3:0/1  ALARM_RESET  "ALARM RESET" %
%   B9:2/9  FT_7000_LOLO_ALT  "FT-7000 LOLO ALERT BIT" %
%   B3:0/0  ALARM_SILENCE  "ALARM SILENCE PUSHBUTTON" %
% Rung: 44 %
SOR GRT N11:10 0 LES F8:5 F10:10 XIO B3:0/1 BST TON T4:10 1.0 0 0 NXB XIC T4:10/DN OSR B3:3/8 OTE B3:3/9 BND EOR
%   N11:10  FT_7000_LOALM_DLY_SP  "FT-7000 LO ALARM DELAY SP FROM HMI" %
%   F8:5  FT_7000_SCI  "FT-7000 SCALED INPUT" %
%   F10:10  FT_7000_LOALM_SP  "FT-7000 LO ALARM SP" %
%   B3:0/1  ALARM_RESET  "ALARM RESET" %
%   T4:10  FT_7000_LOALM_DLY_TM  "FT-7000 LO ALARM DELAY" %
%   B3:3/8  "OSR" %
%   B3:3/9  "FT-7000 LO TRIGGER BIT" %
% Rung: 45 %
SOR BST BST XIC B3:3/9 NXB XIC B9:2/10 XIO B3:0/1 BND OTE B9:2/10 NXB BST XIC B3:3/9 NXB XIC B9:2/11 XIO B3:0/1 XIO B3:0/0 BND OTE B9:2/11 BND EOR
%   B3:3/9  "FT-7000 LO TRIGGER BIT" %
%   B9:2/10  FT_7000_LO_ALM  "FT-7000 LO ALARM BIT" %
%   B3:0/1  ALARM_RESET  "ALARM RESET" %
%   B9:2/11  FT_7000_LO_ALT  "FT-7000 LO ALERT BIT" %
%   B3:0/0  ALARM_SILENCE  "ALARM SILENCE PUSHBUTTON" %
% Rung: 46 %
SOR GRT N11:11 0 GRT F8:5 F10:11 XIO B3:0/1 BST TON T4:11 1.0 0 0 NXB XIC T4:11/DN OSR B3:3/10 OTE B3:3/11 BND EOR
%   N11:11  FT_7000_HIALM_DLY_SP  "FT-7000 HI ALARM DELAY SP FROM HMI" %
%   F8:5  FT_7000_SCI  "FT-7000 SCALED INPUT" %
%   F10:11  FT_7000_HIALM_SP  "FT-7000 HI ALARM SP" %
%   B3:0/1  ALARM_RESET  "ALARM RESET" %
%   T4:11  FT_7000_HIALM_DLY_TM  "FT-7000 HI ALARM DELAY" %
%   B3:3/10  "OSR" %
%   B3:3/11  "FT-7000 HI TRIGGER BIT" %

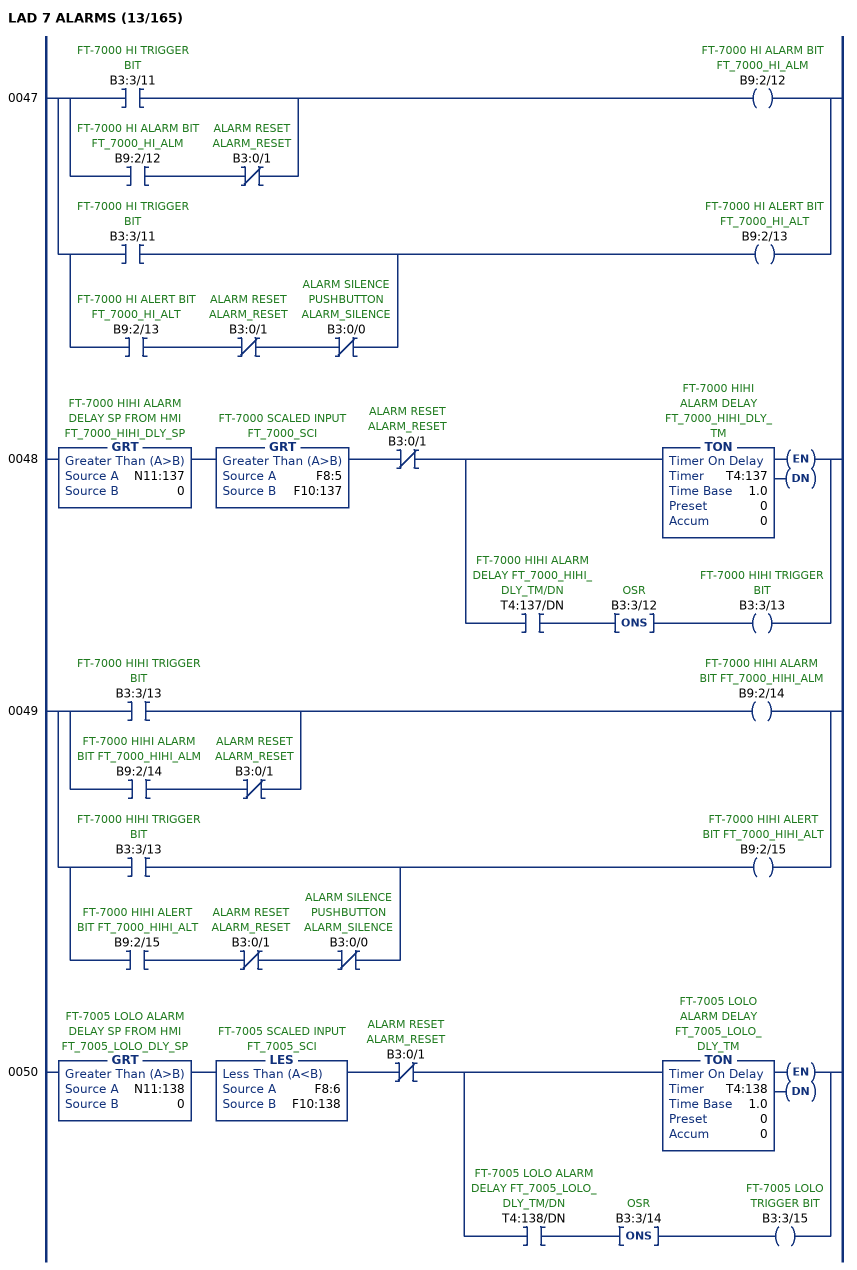
% Rung: 47 %
SOR BST BST XIC B3:3/11 NXB XIC B9:2/12 XIO B3:0/1 BND OTE B9:2/12 NXB BST XIC B3:3/11 NXB XIC B9:2/13 XIO B3:0/1 XIO B3:0/0 BND OTE B9:2/13 BND EOR
%   B3:3/11  "FT-7000 HI TRIGGER BIT" %
%   B9:2/12  FT_7000_HI_ALM  "FT-7000 HI ALARM BIT" %
%   B3:0/1  ALARM_RESET  "ALARM RESET" %
%   B9:2/13  FT_7000_HI_ALT  "FT-7000 HI ALERT BIT" %
%   B3:0/0  ALARM_SILENCE  "ALARM SILENCE PUSHBUTTON" %
% Rung: 48 %
SOR GRT N11:137 0 GRT F8:5 F10:137 XIO B3:0/1 BST TON T4:137 1.0 0 0 NXB XIC T4:137/DN OSR B3:3/12 OTE B3:3/13 BND EOR
%   N11:137  FT_7000_HIHI_DLY_SP  "FT-7000 HIHI ALARM DELAY SP FROM HMI" %
%   F8:5  FT_7000_SCI  "FT-7000 SCALED INPUT" %
%   F10:137  FT_7000_HIHI_SP  "FT-7000 HIHI ALARM SP" %
%   B3:0/1  ALARM_RESET  "ALARM RESET" %
%   T4:137  FT_7000_HIHI_DLY_TM  "FT-7000 HIHI ALARM DELAY" %
%   B3:3/12  "OSR" %
%   B3:3/13  "FT-7000 HIHI TRIGGER BIT" %
% Rung: 49 %
SOR BST BST XIC B3:3/13 NXB XIC B9:2/14 XIO B3:0/1 BND OTE B9:2/14 NXB BST XIC B3:3/13 NXB XIC B9:2/15 XIO B3:0/1 XIO B3:0/0 BND OTE B9:2/15 BND EOR
%   B3:3/13  "FT-7000 HIHI TRIGGER BIT" %
%   B9:2/14  FT_7000_HIHI_ALM  "FT-7000 HIHI ALARM BIT" %
%   B3:0/1  ALARM_RESET  "ALARM RESET" %
%   B9:2/15  FT_7000_HIHI_ALT  "FT-7000 HIHI ALERT BIT" %
%   B3:0/0  ALARM_SILENCE  "ALARM SILENCE PUSHBUTTON" %
% Rung: 50 %
SOR GRT N11:138 0 LES F8:6 F10:138 XIO B3:0/1 BST TON T4:138 1.0 0 0 NXB XIC T4:138/DN OSR B3:3/14 OTE B3:3/15 BND EOR
%   N11:138  FT_7005_LOLO_DLY_SP  "FT-7005 LOLO ALARM DELAY SP FROM HMI" %
%   F8:6  FT_7005_SCI  "FT-7005 SCALED INPUT" %
%   F10:138  FT_7005_LOLO_SP  "FT-7005 LOLO ALARM SP" %
%   B3:0/1  ALARM_RESET  "ALARM RESET" %
%   T4:138  FT_7005_LOLO_DLY_TM  "FT-7005 LOLO ALARM DELAY" %
%   B3:3/14  "OSR" %
%   B3:3/15  "FT-7005 LOLO TRIGGER BIT" %

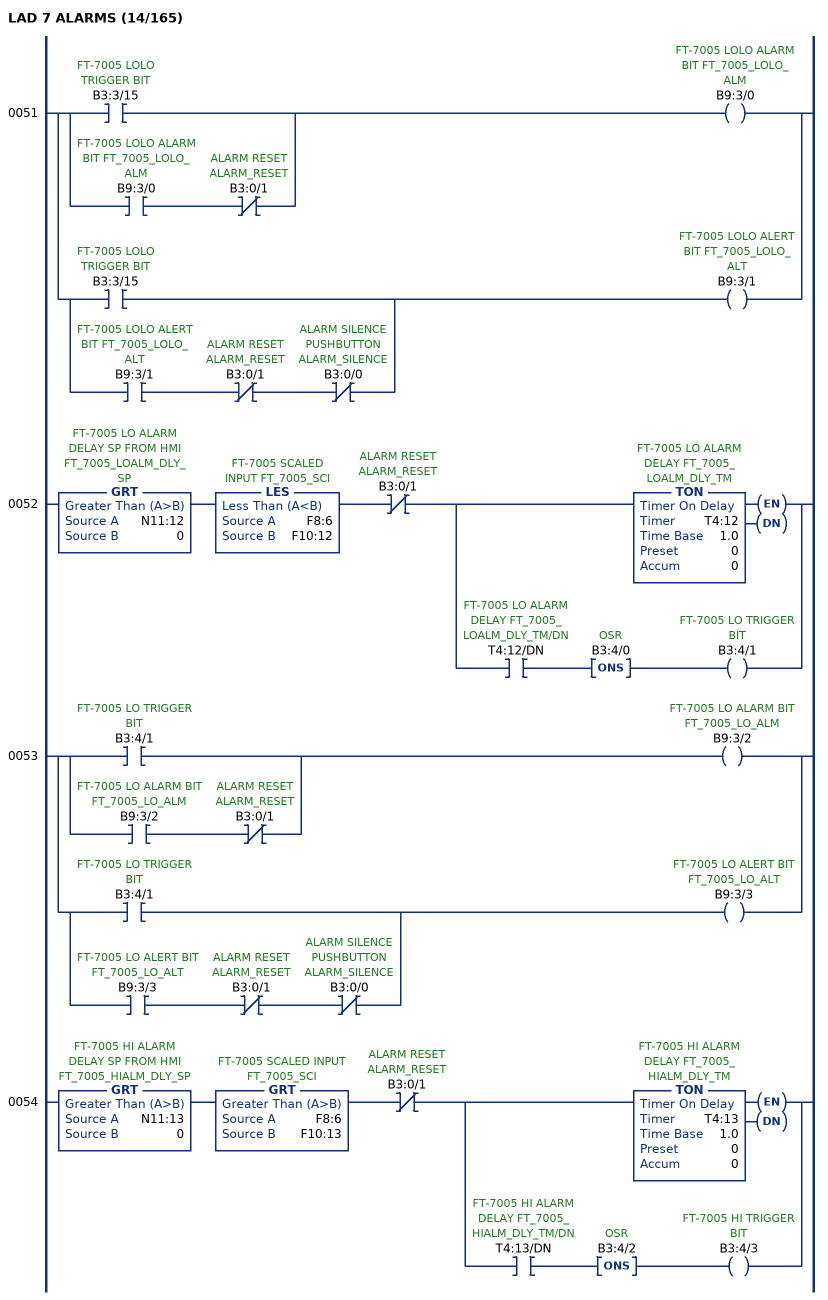
% Rung: 51 %
SOR BST BST XIC B3:3/15 NXB XIC B9:3/0 XIO B3:0/1 BND OTE B9:3/0 NXB BST XIC B3:3/15 NXB XIC B9:3/1 XIO B3:0/1 XIO B3:0/0 BND OTE B9:3/1 BND EOR
%   B3:3/15  "FT-7005 LOLO TRIGGER BIT" %
%   B9:3/0  FT_7005_LOLO_ALM  "FT-7005 LOLO ALARM BIT" %
%   B3:0/1  ALARM_RESET  "ALARM RESET" %
%   B9:3/1  FT_7005_LOLO_ALT  "FT-7005 LOLO ALERT BIT" %
%   B3:0/0  ALARM_SILENCE  "ALARM SILENCE PUSHBUTTON" %
% Rung: 52 %
SOR GRT N11:12 0 LES F8:6 F10:12 XIO B3:0/1 BST TON T4:12 1.0 0 0 NXB XIC T4:12/DN OSR B3:4/0 OTE B3:4/1 BND EOR
%   N11:12  FT_7005_LOALM_DLY_SP  "FT-7005 LO ALARM DELAY SP FROM HMI" %
%   F8:6  FT_7005_SCI  "FT-7005 SCALED INPUT" %
%   F10:12  FT_7005_LOALM_SP  "FT-7005 LO ALARM SP" %
%   B3:0/1  ALARM_RESET  "ALARM RESET" %
%   T4:12  FT_7005_LOALM_DLY_TM  "FT-7005 LO ALARM DELAY" %
%   B3:4/0  "OSR" %
%   B3:4/1  "FT-7005 LO TRIGGER BIT" %
% Rung: 53 %
SOR BST BST XIC B3:4/1 NXB XIC B9:3/2 XIO B3:0/1 BND OTE B9:3/2 NXB BST XIC B3:4/1 NXB XIC B9:3/3 XIO B3:0/1 XIO B3:0/0 BND OTE B9:3/3 BND EOR
%   B3:4/1  "FT-7005 LO TRIGGER BIT" %
%   B9:3/2  FT_7005_LO_ALM  "FT-7005 LO ALARM BIT" %
%   B3:0/1  ALARM_RESET  "ALARM RESET" %
%   B9:3/3  FT_7005_LO_ALT  "FT-7005 LO ALERT BIT" %
%   B3:0/0  ALARM_SILENCE  "ALARM SILENCE PUSHBUTTON" %
% Rung: 54 %
SOR GRT N11:13 0 GRT F8:6 F10:13 XIO B3:0/1 BST TON T4:13 1.0 0 0 NXB XIC T4:13/DN OSR B3:4/2 OTE B3:4/3 BND EOR
%   N11:13  FT_7005_HIALM_DLY_SP  "FT-7005 HI ALARM DELAY SP FROM HMI" %
%   F8:6  FT_7005_SCI  "FT-7005 SCALED INPUT" %
%   F10:13  FT_7005_HIALM_SP  "FT-7005 HI ALARM SP" %
%   B3:0/1  ALARM_RESET  "ALARM RESET" %
%   T4:13  FT_7005_HIALM_DLY_TM  "FT-7005 HI ALARM DELAY" %
%   B3:4/2  "OSR" %
%   B3:4/3  "FT-7005 HI TRIGGER BIT" %

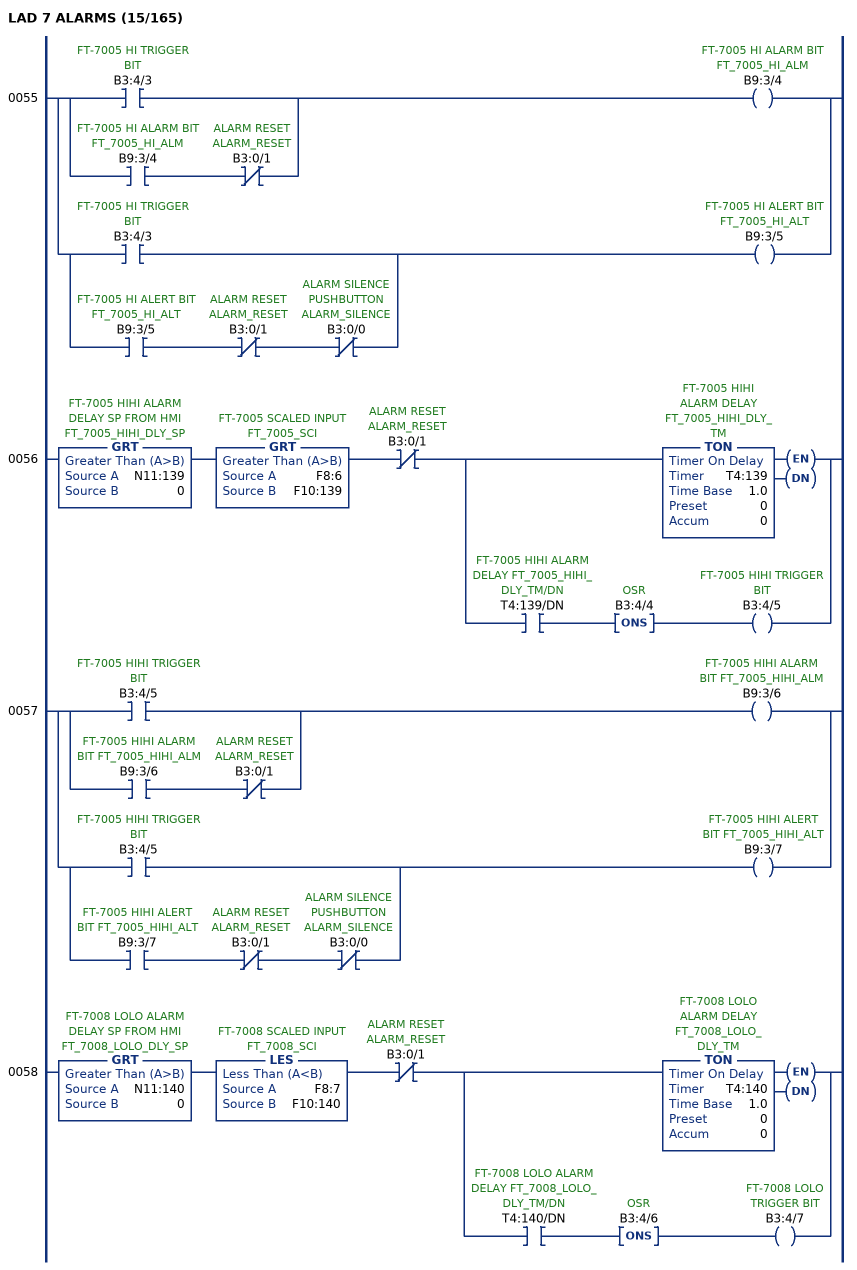
% Rung: 55 %
SOR BST BST XIC B3:4/3 NXB XIC B9:3/4 XIO B3:0/1 BND OTE B9:3/4 NXB BST XIC B3:4/3 NXB XIC B9:3/5 XIO B3:0/1 XIO B3:0/0 BND OTE B9:3/5 BND EOR
%   B3:4/3  "FT-7005 HI TRIGGER BIT" %
%   B9:3/4  FT_7005_HI_ALM  "FT-7005 HI ALARM BIT" %
%   B3:0/1  ALARM_RESET  "ALARM RESET" %
%   B9:3/5  FT_7005_HI_ALT  "FT-7005 HI ALERT BIT" %
%   B3:0/0  ALARM_SILENCE  "ALARM SILENCE PUSHBUTTON" %
% Rung: 56 %
SOR GRT N11:139 0 GRT F8:6 F10:139 XIO B3:0/1 BST TON T4:139 1.0 0 0 NXB XIC T4:139/DN OSR B3:4/4 OTE B3:4/5 BND EOR
%   N11:139  FT_7005_HIHI_DLY_SP  "FT-7005 HIHI ALARM DELAY SP FROM HMI" %
%   F8:6  FT_7005_SCI  "FT-7005 SCALED INPUT" %
%   F10:139  FT_7005_HIHI_SP  "FT-7005 HIHI ALARM SP" %
%   B3:0/1  ALARM_RESET  "ALARM RESET" %
%   T4:139  FT_7005_HIHI_DLY_TM  "FT-7005 HIHI ALARM DELAY" %
%   B3:4/4  "OSR" %
%   B3:4/5  "FT-7005 HIHI TRIGGER BIT" %
% Rung: 57 %
SOR BST BST XIC B3:4/5 NXB XIC B9:3/6 XIO B3:0/1 BND OTE B9:3/6 NXB BST XIC B3:4/5 NXB XIC B9:3/7 XIO B3:0/1 XIO B3:0/0 BND OTE B9:3/7 BND EOR
%   B3:4/5  "FT-7005 HIHI TRIGGER BIT" %
%   B9:3/6  FT_7005_HIHI_ALM  "FT-7005 HIHI ALARM BIT" %
%   B3:0/1  ALARM_RESET  "ALARM RESET" %
%   B9:3/7  FT_7005_HIHI_ALT  "FT-7005 HIHI ALERT BIT" %
%   B3:0/0  ALARM_SILENCE  "ALARM SILENCE PUSHBUTTON" %
% Rung: 58 %
SOR GRT N11:140 0 LES F8:7 F10:140 XIO B3:0/1 BST TON T4:140 1.0 0 0 NXB XIC T4:140/DN OSR B3:4/6 OTE B3:4/7 BND EOR
%   N11:140  FT_7008_LOLO_DLY_SP  "FT-7008 LOLO ALARM DELAY SP FROM HMI" %
%   F8:7  FT_7008_SCI  "FT-7008 SCALED INPUT" %
%   F10:140  FT_7008_LOLO_SP  "FT-7008 LOLO ALARM SP" %
%   B3:0/1  ALARM_RESET  "ALARM RESET" %
%   T4:140  FT_7008_LOLO_DLY_TM  "FT-7008 LOLO ALARM DELAY" %
%   B3:4/6  "OSR" %
%   B3:4/7  "FT-7008 LOLO TRIGGER BIT" %

